// TIA Portal project "Sirius" (V17)

(* hardware
DEVICE "S7-1200 station_1"  S7-1200 Station
   slot 0: "Rack_0"  S7-1200 Rack  Rack  V1.0
   slot 1: "PLC_1"  CPU 1214C DC/DC/DC  6ES7 214-1AG40-0XB0  V4.5
   slot 2: "DI 16x24VDC/DQ 16xRelay_1"  SM 1223 DI16/DQ16 x relay  6ES7 223-1PL32-0XB0  V2.0
   slot 3: "DI 8/DQ 8x24VDC_1"  6ES7 223-1BH32-0XB0  V2.0
   slot 4: "AI 8x13BIT_1"  6ES7 231-4HF32-0XB0  V2.1
   slot 5: "AI 4x13BIT_1"  6ES7 231-4HD32-0XB0  V2.1
   slot 101: "CM 1241 (RS422/485)_1"  6ES7 241-1CH32-0XB0  V2.2
   slot 102: "CM 1241 (RS422/485)_2"  6ES7 241-1CH32-0XB0  V2.2
*)

// ===== PLC "PLC_1"  CPU 1214C DC/DC/DC =====

VAR_GLOBAL   // PLC tag table "Default tag table"
   "System_Byte" AT %MB1 : Byte;
   "FirstScan" AT %M1.0 : Bool;
   "DiagStatusUpdate" AT %M1.1 : Bool;
   "AlwaysTRUE" AT %M1.2 : Bool;
   "AlwaysFALSE" AT %M1.3 : Bool;
   "Clock_Byte" AT %MB0 : Byte;
   "Clock_10Hz" AT %M0.0 : Bool;
   "Clock_5Hz" AT %M0.1 : Bool;
   "Clock_2.5Hz" AT %M0.2 : Bool;
   "Clock_2Hz" AT %M0.3 : Bool;
   "Clock_1.25Hz" AT %M0.4 : Bool;
   "Clock_1Hz" AT %M0.5 : Bool;
   "Clock_0.625Hz" AT %M0.6 : Bool;
   "Clock_0.5Hz" AT %M0.7 : Bool;
END_VAR

VAR_GLOBAL   // PLC tag table "DI"
   "DIa1.0" AT %I0.0 : Bool;   // Наличие напряжения на основном вводе
   "DIa1.1" AT %I0.1 : Bool;   // Наличие напряжения на резервном вводе
   "DIa1.2" AT %I0.2 : Bool;   // Наличие питания 220В внешних потр.
   "DIa1.3" AT %I0.3 : Bool;   // Наличие пит. 220В собств. нужд; Питание 24В от АКБ
   "DIa1.4" AT %I0.4 : Bool;   // АКБ разряжена
   "DIa1.5" AT %I0.5 : Bool;   // Отключение звука
   "DIa1.6" AT %I0.6 : Bool;   // Стоп АН
   "DIa1.7" AT %I0.7 : Bool;   // Автоматическое управление
   "DIb1.0" AT %I1.0 : Bool;   // Ручное управление
   "DIb1.1" AT %I1.1 : Bool;   // Тест индикации
   "DIb1.2" AT %I1.2 : Bool;   // Затопление
   "DIb1.3" AT %I1.3 : Bool;   // Открытие двери
   "reserved_DIb1.4" AT %I1.4 : Bool;   // --------
   "reserved_DIb1.5" AT %I1.5 : Bool;   // --------
   "DIa2.0" AT %I8.0 : Bool;   // Авт. выкл. НБ № 1 включен
   "DIa2.1" AT %I8.1 : Bool;   // Контактор НБ № 1 вклюен
   "DIa2.2" AT %I8.2 : Bool;   // Авт. выкл. НБ № 2 включен
   "DIa2.3" AT %I8.3 : Bool;   // Контактор НБ № 2 включен
   "DIa2.4" AT %I8.4 : Bool;   // Авт. выкл. НБ № 3 включен
   "DIa2.5" AT %I8.5 : Bool;   // Контактор НБ № 3 включен
   "DIa2.6" AT %I8.6 : Bool;   // Авт. выкл. НБ № 4 включен
   "DIa2.7" AT %I8.7 : Bool;   // Контактор НБ № 4 включен
   "DIb2.0" AT %I9.0 : Bool;   // Авт. выкл. НБ № 5 включен
   "DIb2.1" AT %I9.1 : Bool;   // Контактор НБ № 5 включен
   "DIb2.2" AT %I9.2 : Bool;   // Авт. выкл. НП включен
   "DIb2.3" AT %I9.3 : Bool;   // Контактор НП включен
   "reserved_DIb2.4" AT %I9.4 : Bool;   // --------
   "reserved_DIb2.5" AT %I9.5 : Bool;   // --------
   "reserved_DIb2.6" AT %I9.6 : Bool;   // --------
   "reserved_DIb2.7" AT %I9.7 : Bool;   // --------
   "DIa3.0" AT %I12.0 : Bool;   // УУС.1: Проток
   "DIa3.1" AT %I12.1 : Bool;   // УУС.2: Проток
   "DIa3.2" AT %I12.2 : Bool;   // УУС.3: Проток
   "DIa3.3" AT %I12.3 : Bool;   // УУС.4: Проток
   "reserved_DIa3.4" AT %I12.4 : Bool;   // --------
   "reserved_DIa3.5" AT %I12.5 : Bool;   // --------
   "reserved_DIa3.6" AT %I12.6 : Bool;   // --------
   "reserved_DIa3.7" AT %I12.7 : Bool;   // --------
END_VAR

VAR_GLOBAL   // PLC tag table "DQ"
   "DQa1.0" AT %Q0.0 : Bool;   // Пожар
   "DQa1.1" AT %Q0.1 : Bool;   // Пуск насосного агрегата
   "DQa1.2" AT %Q0.2 : Bool;   // Отсутствие неисправности
   "DQa1.3" AT %Q0.3 : Bool;   // Автоматика отключена
   "DQa1.4" AT %Q0.4 : Bool;   // Дежурный режим
   "DQa1.5" AT %Q0.5 : Bool;   // Звуковой сигнал
   "DQa1.6" AT %Q0.6 : Bool;   // Система отключена
   "DQa1.7" AT %Q0.7 : Bool;   // Звук отключен
   "reserved_DQb1.0" AT %Q1.0 : Bool;   // -----
   "reserved_DQb1.1" AT %Q1.1 : Bool;   // -----
   "RQa2.0" AT %Q8.0 : Bool;   // Управление НБ № 1
   "RQa2.1" AT %Q8.1 : Bool;   // Управление НБ № 2
   "RQa2.2" AT %Q8.2 : Bool;   // Управление НБ № 3
   "RQa2.3" AT %Q8.3 : Bool;   // Управление НБ № 4
   "RQa2.4" AT %Q8.4 : Bool;   // Управление НБ № 5
   "RQa2.5" AT %Q8.5 : Bool;   // Управление НП
   "reserved_RQa2.6" AT %Q8.6 : Bool;   // -----
   "reserved_RQa2.7" AT %Q8.7 : Bool;   // -----
   "RQb2.0" AT %Q9.0 : Bool;   // Неисправность НБ № 1
   "RQb2.1" AT %Q9.1 : Bool;   // Неисправность НБ № 2
   "RQb2.2" AT %Q9.2 : Bool;   // Неисправность НБ № 3
   "RQb2.3" AT %Q9.3 : Bool;   // Неисправность НБ № 4
   "RQb2.4" AT %Q9.4 : Bool;   // Неисправность НБ № 5
   "RQb2.5" AT %Q9.5 : Bool;   // Неисправность НП
   "reserved_RQb2.6" AT %Q9.6 : Bool;   // -----
   "reserved_RQb2.7" AT %Q9.7 : Bool;   // -----
   "DQa3.0" AT %Q12.0 : Bool;   // УУС.1: Срабатывание
   "DQa3.1" AT %Q12.1 : Bool;   // УУС.1: Неисправность
   "DQa3.2" AT %Q12.2 : Bool;   // УУС.2: Срабатывание
   "DQa3.3" AT %Q12.3 : Bool;   // УУС.2: Неисправность
   "DQa3.4" AT %Q12.4 : Bool;   // УУС.3: Срабатывание
   "DQa3.5" AT %Q12.5 : Bool;   // УУС.3: Неисправность
   "DQa3.6" AT %Q12.6 : Bool;   // УУС.4: Срабатывание
   "DQa3.7" AT %Q12.7 : Bool;   // УУС.4: Неисправность
END_VAR

VAR_GLOBAL   // PLC tag table "AI"
   "AI4.0" AT %IW144 : Int;   // Датчик низкого давления PIS1.1
   "AI4.1" AT %IW146 : Int;   // Датчик низкого давления PIS1.2
   "AI4.2" AT %IW148 : Int;   // Датчик высокого давления PIS2.1
   "AI4.3" AT %IW150 : Int;   // Датчик высокого давления PIS2.2
   "AI4.4" AT %IW152 : Int;   // Датчик давления НБ №1
   "AI4.5" AT %IW154 : Int;   // Датчик давления НБ №2
   "AI4.6" AT %IW156 : Int;   // Датчик давления НБ №3
   "AI4.7" AT %IW158 : Int;   // Датчик давления НБ №4
   "AI5.0" AT %IW160 : Int;   // Датчик давления НБ №5
   "reserved_AI5.1" AT %IW162 : Int;   // ------
   "reserved_AI5.2" AT %IW164 : Int;   // ------
   "reserved_AI5.3" AT %IW166 : Int;   // ------
END_VAR

VAR_GLOBAL   // PLC tag table "MODBUS"
   "MB_MODE_auto" AT %M4002.1 : Bool;
   "MB_MODE_manual" AT %M4002.2 : Bool;
   "MB_MODE_blocked" AT %M4002.3 : Bool;
   "MB_MODE_standby" AT %M4002.4 : Bool;
   "MB_MODE_standby_pressure_high" AT %M4002.5 : Bool;
   "MB_BUTTON_Global_Stop" AT %M4002.6 : Bool;
   "MB_Global_Stop" AT %M4002.7 : Bool;
   "MB_BUTTON_Sound_Off" AT %M4003.0 : Bool;
   "MB_BUTTON_Led_Test" AT %M4003.1 : Bool;
   "MB_STATE_380_main" AT %M4003.2 : Bool;
   "MB_STATE_380_backup" AT %M4003.3 : Bool;
   "MB_STATE_220_inner" AT %M4003.4 : Bool;
   "MB_STATE_220_outer" AT %M4003.5 : Bool;
   "MB_STATE_door_opened" AT %M4003.6 : Bool;
   "MB_ERROR_underwater" AT %M4003.7 : Bool;
   "MB_ERROR_no_water" AT %M4004.0 : Bool;
   "MB_ERROR_no_water_fire" AT %M4004.1 : Bool;
   "MB_ERROR_inlet_pressure_low" AT %M4004.2 : Bool;
   "MB_ERROR_global" AT %M4004.3 : Bool;
   "MB_ERROR_Main_Ball_Valves" AT %M4004.4 : Bool;
   "MB_ERROR_BALL_VALVE_ANY" AT %M4004.5 : Bool;
   "MB_ERROR_any" AT %M4004.6 : Bool;
   "MB_SIGNAL_fire" AT %M4004.7 : Bool;
   "MB_SIGNAL_fire_by_pressure" AT %M4005.0 : Bool;
   "MB_ERROR_high_pressure_redundancy" AT %M4005.1 : Bool;
   "MB_ERROR_low_pressure_redundancy" AT %M4005.2 : Bool;
   "MB_SIGNAL_first_pump_has_started" AT %M4005.3 : Bool;
   "MB_Start_standby_pump" AT %M4005.4 : Bool;
   "MB_Secret_condition" AT %M4005.5 : Bool;
   "MB_ERROR_Battery_low" AT %M4005.6 : Bool;
   "MB_ERROR_connection_lost" AT %M4005.7 : Bool;
   "MB_ERROR_connection_lost_TOF" AT %M4006.0 : Bool;
   "MB_ERROR_connection_lost_TON" AT %M4006.1 : Bool;
   "MB_SENSOR_low_pressure_PIS1.1_error" AT %M4006.2 : Bool;
   "MB_SENSOR_low_pressure_PIS1.2_error" AT %M4006.3 : Bool;
   "MB_SENSOR_high_pressure_PIS2.1_error" AT %M4006.4 : Bool;
   "MB_SENSOR_high_pressure_PIS2.2_error" AT %M4006.5 : Bool;
   "MB_IN_valve_gate__ERROR_B1" AT %M4006.6 : Bool;
   "MB_IN_valve_gate__ERROR_B2" AT %M4006.7 : Bool;
   "MB_IN_valve_gate__ERROR_B3" AT %M4007.0 : Bool;
   "MB_IN_valve_gate__ERROR_B4" AT %M4007.1 : Bool;
   "MB_IN_valve_gate__ERROR_B5" AT %M4007.2 : Bool;
   "MB_IN_valve_gate__ERROR_B6" AT %M4007.3 : Bool;
   "MB_IN_valve_gate__ERROR_B7" AT %M4007.4 : Bool;
   "MB_IN_valve_gate__ERROR_B8" AT %M4007.5 : Bool;
   "MB_IN_valve_gate__ERROR_B9" AT %M4007.6 : Bool;
   "MB_ERROR_IN_VALVE_ANY" AT %M4007.7 : Bool;
   "MB_SENSOR_flow_UUS1" AT %M4008.0 : Bool;
   "MB_SENSOR_flow_UUS2" AT %M4008.1 : Bool;
   "MB_SENSOR_flow_UUS3" AT %M4008.2 : Bool;
   "MB_SENSOR_flow_UUS4" AT %M4008.3 : Bool;
   "MB_ERROR_UUS1" AT %M4008.4 : Bool;
   "MB_ERROR_UUS2" AT %M4008.5 : Bool;
   "MB_ERROR_UUS3" AT %M4008.6 : Bool;
   "MB_ERROR_UUS4" AT %M4008.7 : Bool;
   "MB_ERROR_UUS_ANY" AT %M4009.0 : Bool;
   "MB_ERROR_UUS_ALL" AT %M4009.1 : Bool;
   "MB_State_switch_pump1" AT %M4009.2 : Bool;
   "MB_State_switch_pump2" AT %M4009.3 : Bool;
   "MB_State_switch_pump3" AT %M4009.4 : Bool;
   "MB_State_switch_pump4" AT %M4009.5 : Bool;
   "MB_State_switch_pump5" AT %M4009.6 : Bool;
   "MB_Error_pump1" AT %M4009.7 : Bool;
   "MB_Error_pump2" AT %M4010.0 : Bool;
   "MB_Error_pump3" AT %M4010.1 : Bool;
   "MB_Error_pump4" AT %M4010.2 : Bool;
   "MB_Error_pump5" AT %M4010.3 : Bool;
   "MB_State_starter_pump1" AT %M4010.4 : Bool;
   "MB_State_starter_pump2" AT %M4010.5 : Bool;
   "MB_State_starter_pump3" AT %M4010.6 : Bool;
   "MB_State_starter_pump4" AT %M4010.7 : Bool;
   "MB_State_starter_pump5" AT %M4011.0 : Bool;
   "MB_State_work_pump1" AT %M4011.1 : Bool;
   "MB_State_work_pump2" AT %M4011.2 : Bool;
   "MB_State_work_pump3" AT %M4011.3 : Bool;
   "MB_State_work_pump4" AT %M4011.4 : Bool;
   "MB_State_work_pump5" AT %M4011.5 : Bool;
   "MB_Pump_pressure_sensor_error1" AT %M4011.6 : Bool;
   "MB_Pump_pressure_sensor_error2" AT %M4011.7 : Bool;
   "MB_Pump_pressure_sensor_error3" AT %M4012.0 : Bool;
   "MB_Pump_pressure_sensor_error4" AT %M4012.1 : Bool;
   "MB_Pump_pressure_sensor_error5" AT %M4012.2 : Bool;
   "MB_State_switch_standby_pump" AT %M4012.3 : Bool;
   "MB_Error_any_pump" AT %M4012.4 : Bool;
   "MB_Error_standby_pump" AT %M4012.5 : Bool;
   "MB_State_starter_standby_pump" AT %M4012.6 : Bool;
   "MB_State_work_standby_pump" AT %M4012.7 : Bool;
   "MB_State_work_any_pump" AT %M4013.0 : Bool;
   "MB_ERROR_PUMPS_ANY" AT %M4013.1 : Bool;
   "MB_ERROR_PUMPS_ALL" AT %M4013.2 : Bool;
   "MB_Low_pressure_valve_B1_open_OFF" AT %M4013.3 : Bool;
   "MB_Low_pressure_valve_B1_open_NO_signal" AT %M4013.4 : Bool;
   "MB_Low_pressure_valve_B1_open_short" AT %M4013.5 : Bool;
   "MB_Low_pressure_valve_B1_open_brake" AT %M4013.6 : Bool;
   "MB_Low_pressure_valve_B1_open_Signal" AT %M4013.7 : Bool;
   "MB_Low_pressure_valve_B1_close_OFF" AT %M4014.0 : Bool;
   "MB_Low_pressure_valve_B1_close_NO_signal" AT %M4014.1 : Bool;
   "MB_Low_pressure_valve_B1_close_short" AT %M4014.2 : Bool;
   "MB_Low_pressure_valve_B1_close_brake" AT %M4014.3 : Bool;
   "MB_Low_pressure_valve_B1_close_Signal" AT %M4014.4 : Bool;
   "MB_Low_pressure_valve_B2_open_OFF" AT %M4014.5 : Bool;
   "MB_Low_pressure_valve_B2_open_NO_signal" AT %M4014.6 : Bool;
   "MB_Low_pressure_valve_B2_open_short" AT %M4014.7 : Bool;
   "MB_Low_pressure_valve_B2_open_brake" AT %M4015.0 : Bool;
   "MB_Low_pressure_valve_B2_open_Signal" AT %M4015.1 : Bool;
   "MB_Low_pressure_valve_B2_close_OFF" AT %M4015.2 : Bool;
   "MB_Low_pressure_valve_B2_close_NO_signal" AT %M4015.3 : Bool;
   "MB_Low_pressure_valve_B2_close_short" AT %M4015.4 : Bool;
   "MB_Low_pressure_valve_B2_close_brake" AT %M4015.5 : Bool;
   "MB_Low_pressure_valve_B2_close_Signal" AT %M4015.6 : Bool;
   "MB_Low_pressure_valve_B3_open_OFF" AT %M4015.7 : Bool;
   "MB_Low_pressure_valve_B3_open_NO_signal" AT %M4016.0 : Bool;
   "MB_Low_pressure_valve_B3_open_short" AT %M4016.1 : Bool;
   "MB_Low_pressure_valve_B3_open_brake" AT %M4016.2 : Bool;
   "MB_Low_pressure_valve_B3_open_Signal" AT %M4016.3 : Bool;
   "MB_Low_pressure_valve_B3_close_OFF" AT %M4016.4 : Bool;
   "MB_Low_pressure_valve_B3_close_NO_signal" AT %M4016.5 : Bool;
   "MB_Low_pressure_valve_B3_close_short" AT %M4016.6 : Bool;
   "MB_Low_pressure_valve_B3_close_brake" AT %M4016.7 : Bool;
   "MB_Low_pressure_valve_B3_close_Signal" AT %M4017.0 : Bool;
   "MB_Low_pressure_valve_B4_open_OFF" AT %M4017.1 : Bool;
   "MB_Low_pressure_valve_B4_open_NO_signal" AT %M4017.2 : Bool;
   "MB_Low_pressure_valve_B4_open_short" AT %M4017.3 : Bool;
   "MB_Low_pressure_valve_B4_open_brake" AT %M4017.4 : Bool;
   "MB_Low_pressure_valve_B4_open_Signal" AT %M4017.5 : Bool;
   "MB_Low_pressure_valve_B4_close_OFF" AT %M4017.6 : Bool;
   "MB_Low_pressure_valve_B4_close_NO_signal" AT %M4017.7 : Bool;
   "MB_Low_pressure_valve_B4_close_short" AT %M4018.0 : Bool;
   "MB_Low_pressure_valve_B4_close_brake" AT %M4018.1 : Bool;
   "MB_Low_pressure_valve_B4_close_Signal" AT %M4018.2 : Bool;
   "MB_Low_pressure_valve_B5_open_OFF" AT %M4018.3 : Bool;
   "MB_Low_pressure_valve_B5_open_NO_signal" AT %M4018.4 : Bool;
   "MB_Low_pressure_valve_B5_open_short" AT %M4018.5 : Bool;
   "MB_Low_pressure_valve_B5_open_brake" AT %M4018.6 : Bool;
   "MB_Low_pressure_valve_B5_open_Signal" AT %M4018.7 : Bool;
   "MB_Low_pressure_valve_B5_close_OFF" AT %M4019.0 : Bool;
   "MB_Low_pressure_valve_B5_close_NO_signal" AT %M4019.1 : Bool;
   "MB_Low_pressure_valve_B5_close_short" AT %M4019.2 : Bool;
   "MB_Low_pressure_valve_B5_close_brake" AT %M4019.3 : Bool;
   "MB_Low_pressure_valve_B5_close_Signal" AT %M4019.4 : Bool;
   "MB_Low_pressure_valve_B6_open_OFF" AT %M4019.5 : Bool;
   "MB_Low_pressure_valve_B6_open_NO_signal" AT %M4019.6 : Bool;
   "MB_Low_pressure_valve_B6_open_short" AT %M4019.7 : Bool;
   "MB_Low_pressure_valve_B6_open_brake" AT %M4020.0 : Bool;
   "MB_Low_pressure_valve_B6_open_Signal" AT %M4020.1 : Bool;
   "MB_Low_pressure_valve_B6_close_OFF" AT %M4020.2 : Bool;
   "MB_Low_pressure_valve_B6_close_NO_signal" AT %M4020.3 : Bool;
   "MB_Low_pressure_valve_B6_close_short" AT %M4020.4 : Bool;
   "MB_Low_pressure_valve_B6_close_brake" AT %M4020.5 : Bool;
   "MB_Low_pressure_valve_B6_close_Signal" AT %M4020.6 : Bool;
   "MB_Low_pressure_valve_B7_open_OFF" AT %M4020.7 : Bool;
   "MB_Low_pressure_valve_B7_open_NO_signal" AT %M4021.0 : Bool;
   "MB_Low_pressure_valve_B7_open_short" AT %M4021.1 : Bool;
   "MB_Low_pressure_valve_B7_open_brake" AT %M4021.2 : Bool;
   "MB_Low_pressure_valve_B7_open_Signal" AT %M4021.3 : Bool;
   "MB_Low_pressure_valve_B7_close_OFF" AT %M4021.4 : Bool;
   "MB_Low_pressure_valve_B7_close_NO_signal" AT %M4021.5 : Bool;
   "MB_Low_pressure_valve_B7_close_short" AT %M4021.6 : Bool;
   "MB_Low_pressure_valve_B7_close_brake" AT %M4021.7 : Bool;
   "MB_Low_pressure_valve_B7_close_Signal" AT %M4022.0 : Bool;
   "MB_Low_pressure_valve_B8_open_OFF" AT %M4022.1 : Bool;
   "MB_Low_pressure_valve_B8_open_NO_signal" AT %M4022.2 : Bool;
   "MB_Low_pressure_valve_B8_open_short" AT %M4022.3 : Bool;
   "MB_Low_pressure_valve_B8_open_brake" AT %M4022.4 : Bool;
   "MB_Low_pressure_valve_B8_open_Signal" AT %M4022.5 : Bool;
   "MB_Low_pressure_valve_B8_close_OFF" AT %M4022.6 : Bool;
   "MB_Low_pressure_valve_B8_close_NO_signal" AT %M4022.7 : Bool;
   "MB_Low_pressure_valve_B8_close_short" AT %M4023.0 : Bool;
   "MB_Low_pressure_valve_B8_close_brake" AT %M4023.1 : Bool;
   "MB_Low_pressure_valve_B8_close_Signal" AT %M4023.2 : Bool;
   "MB_Low_pressure_valve_B9_open_OFF" AT %M4023.3 : Bool;
   "MB_Low_pressure_valve_B9_open_NO_signal" AT %M4023.4 : Bool;
   "MB_Low_pressure_valve_B9_open_short" AT %M4023.5 : Bool;
   "MB_Low_pressure_valve_B9_open_brake" AT %M4023.6 : Bool;
   "MB_Low_pressure_valve_B9_open_Signal" AT %M4023.7 : Bool;
   "MB_Low_pressure_valve_B9_close_OFF" AT %M4024.0 : Bool;
   "MB_Low_pressure_valve_B9_close_NO_signal" AT %M4024.1 : Bool;
   "MB_Low_pressure_valve_B9_close_short" AT %M4024.2 : Bool;
   "MB_Low_pressure_valve_B9_close_brake" AT %M4024.3 : Bool;
   "MB_Low_pressure_valve_B9_close_Signal" AT %M4024.4 : Bool;
   "MB_Ball_valve_K38.1_open_OFF" AT %M4024.5 : Bool;
   "MB_Ball_valve_K38.1_open_NO_signal" AT %M4024.6 : Bool;
   "MB_Ball_valve_K38.1_open_short" AT %M4024.7 : Bool;
   "MB_Ball_valve_K38.1_open_brake" AT %M4025.0 : Bool;
   "MB_Ball_valve_K38.1_open_Signal" AT %M4025.1 : Bool;
   "MB_Ball_valve_K38.2_open_OFF" AT %M4025.2 : Bool;
   "MB_Ball_valve_K38.2_open_NO_signal" AT %M4025.3 : Bool;
   "MB_Ball_valve_K38.2_open_short" AT %M4025.4 : Bool;
   "MB_Ball_valve_K38.2_open_brake" AT %M4025.5 : Bool;
   "MB_Ball_valve_K38.2_open_Signal" AT %M4025.6 : Bool;
   "MB_Ball_valve_K38.3_open_OFF" AT %M4025.7 : Bool;
   "MB_Ball_valve_K38.3_open_NO_signal" AT %M4026.0 : Bool;
   "MB_Ball_valve_K38.3_open_short" AT %M4026.1 : Bool;
   "MB_Ball_valve_K38.3_open_brake" AT %M4026.2 : Bool;
   "MB_Ball_valve_K38.3_open_Signal" AT %M4026.3 : Bool;
   "MB_Ball_valve_K38.4_open_OFF" AT %M4026.4 : Bool;
   "MB_Ball_valve_K38.4_open_NO_signal" AT %M4026.5 : Bool;
   "MB_Ball_valve_K38.4_open_short" AT %M4026.6 : Bool;
   "MB_Ball_valve_K38.4_open_brake" AT %M4026.7 : Bool;
   "MB_Ball_valve_K38.4_open_Signal" AT %M4027.0 : Bool;
   "MB_Ball_valve_K38.5_open_OFF" AT %M4027.1 : Bool;
   "MB_Ball_valve_K38.5_open_NO_signal" AT %M4027.2 : Bool;
   "MB_Ball_valve_K38.5_open_short" AT %M4027.3 : Bool;
   "MB_Ball_valve_K38.5_open_brake" AT %M4027.4 : Bool;
   "MB_Ball_valve_K38.5_open_Signal" AT %M4027.5 : Bool;
   "MB_UUS.1_open_OFF" AT %M4027.6 : Bool;
   "MB_UUS.1_open_NO_signal" AT %M4027.7 : Bool;
   "MB_UUS.1_open_short" AT %M4028.0 : Bool;
   "MB_UUS.1_open_brake" AT %M4028.1 : Bool;
   "MB_UUS.1_open_Signal" AT %M4028.2 : Bool;
   "MB_UUS.2_open_OFF" AT %M4028.3 : Bool;
   "MB_UUS.2_open_NO_signal" AT %M4028.4 : Bool;
   "MB_UUS.2_open_short" AT %M4028.5 : Bool;
   "MB_UUS.2_open_brake" AT %M4028.6 : Bool;
   "MB_UUS.2_open_Signal" AT %M4028.7 : Bool;
   "MB_UUS.3_open_OFF" AT %M4029.0 : Bool;
   "MB_UUS.3_open_NO_signal" AT %M4029.1 : Bool;
   "MB_UUS.3_open_short" AT %M4029.2 : Bool;
   "MB_UUS.3_open_brake" AT %M4029.3 : Bool;
   "MB_UUS.3_open_Signal" AT %M4029.4 : Bool;
   "MB_UUS.4_open_OFF" AT %M4029.5 : Bool;
   "MB_UUS.4_open_NO_signal" AT %M4029.6 : Bool;
   "MB_UUS.4_open_short" AT %M4029.7 : Bool;
   "MB_UUS.4_open_brake" AT %M4030.0 : Bool;
   "MB_UUS.4_open_Signal" AT %M4030.1 : Bool;
   "MB_SENSOR_low_pressure_PIS1.1" AT %MD4032 : Real;
   "MB_SENSOR_low_pressure_PIS1.2" AT %MD4036 : Real;
   "MB_SENSOR_high_pressure_PIS2.1" AT %MD4040 : Real;
   "MB_SENSOR_high_pressure_PIS2.2" AT %MD4044 : Real;
   "MB_INDICATION_high_pressure" AT %MD4048 : Real;
   "MB_INDICATION_low_pressure" AT %MD4052 : Real;
   "MB_Pump_pressure_sensor1" AT %MD4056 : Real;
   "MB_Pump_pressure_sensor2" AT %MD4060 : Real;
   "MB_Pump_pressure_sensor3" AT %MD4064 : Real;
   "MB_Pump_pressure_sensor4" AT %MD4068 : Real;
   "MB_Pump_pressure_sensor5" AT %MD4072 : Real;
   "MB_BUTTON_START_KPPU" AT %M4000.0 : Bool;
   "MB_BUTTON_STOP_KPPU" AT %M4000.1 : Bool;
   "MB_KPPU_connection_test" AT %M4000.2 : Bool;
   "MB_PPU_connection_test" AT %M4002.0 : Bool;
END_VAR

VAR_GLOBAL   // PLC tag table "HMI"
   "HMI_BUTTON_START_KPPU" AT %M600.0 : Bool;
   "HMI_BUTTON_STOP_KPPU" AT %M600.1 : Bool;
   "HMI_MODE_auto" AT %M600.2 : Bool;
   "HMI_MODE_manual" AT %M600.3 : Bool;
   "HMI_MODE_blocked" AT %M600.4 : Bool;
   "HMI_MODE_standby" AT %M600.5 : Bool;
   "HMI_MODE_standby_pressure_high" AT %M600.6 : Bool;
   "HMI_BUTTON_Global_Stop" AT %M600.7 : Bool;
   "HMI_Global_Stop" AT %M601.0 : Bool;
   "HMI_BUTTON_Sound_Off" AT %M601.1 : Bool;
   "HMI_BUTTON_Led_Test" AT %M601.2 : Bool;
   "HMI_STATE_380_main" AT %M601.3 : Bool;
   "HMI_STATE_380_backup" AT %M601.4 : Bool;
   "HMI_STATE_220_inner" AT %M601.5 : Bool;
   "HMI_STATE_220_outer" AT %M601.6 : Bool;
   "HMI_STATE_door_opened" AT %M601.7 : Bool;
   "HMI_ERROR_underwater" AT %M602.0 : Bool;
   "HMI_ERROR_no_water" AT %M602.1 : Bool;
   "HMI_ERROR_no_water_fire" AT %M602.2 : Bool;
   "HMI_ERROR_inlet_pressure_low" AT %M602.3 : Bool;
   "HMI_ERROR_global" AT %M602.4 : Bool;
   "HMI_ERROR_Main_Ball_Valves" AT %M602.5 : Bool;
   "HMI_ERROR_BALL_VALVE_ANY" AT %M602.6 : Bool;
   "HMI_ERROR_any" AT %M602.7 : Bool;
   "HMI_SIGNAL_fire" AT %M603.0 : Bool;
   "HMI_SIGNAL_fire_by_pressure" AT %M603.1 : Bool;
   "HMI_ERROR_high_pressure_redundancy" AT %M603.2 : Bool;
   "HMI_ERROR_low_pressure_redundancy" AT %M603.3 : Bool;
   "HMI_SIGNAL_first_pump_has_started" AT %M603.4 : Bool;
   "HMI_Start_standby_pump" AT %M603.5 : Bool;
   "HMI_Secret_condition" AT %M603.6 : Bool;
   "HMI_ERROR_Battery_low" AT %M603.7 : Bool;
   "HMI_ERROR_connection_lost" AT %M604.0 : Bool;
   "HMI_ERROR_connection_lost_TOF" AT %M604.1 : Bool;
   "HMI_ERROR_connection_lost_TON" AT %M604.2 : Bool;
   "HMI_SENSOR_low_pressure_PIS1.1_error" AT %M604.3 : Bool;
   "HMI_SENSOR_low_pressure_PIS1.2_error" AT %M604.4 : Bool;
   "HMI_SENSOR_high_pressure_PIS2.1_error" AT %M604.5 : Bool;
   "HMI_SENSOR_high_pressure_PIS2.2_error" AT %M604.6 : Bool;
   "HMI_IN_valve_gate__ERROR_B1" AT %M604.7 : Bool;
   "HMI_IN_valve_gate__ERROR_B2" AT %M605.0 : Bool;
   "HMI_IN_valve_gate__ERROR_B3" AT %M605.1 : Bool;
   "HMI_IN_valve_gate__ERROR_B4" AT %M605.2 : Bool;
   "HMI_IN_valve_gate__ERROR_B5" AT %M605.3 : Bool;
   "HMI_IN_valve_gate__ERROR_B6" AT %M605.4 : Bool;
   "HMI_IN_valve_gate__ERROR_B7" AT %M605.5 : Bool;
   "HMI_IN_valve_gate__ERROR_B8" AT %M605.6 : Bool;
   "HMI_IN_valve_gate__ERROR_B9" AT %M605.7 : Bool;
   "HMI_ERROR_IN_VALVE_ANY" AT %M606.0 : Bool;
   "HMI_SENSOR_flow_UUS1" AT %M606.1 : Bool;
   "HMI_SENSOR_flow_UUS2" AT %M606.2 : Bool;
   "HMI_SENSOR_flow_UUS3" AT %M606.3 : Bool;
   "HMI_SENSOR_flow_UUS4" AT %M606.4 : Bool;
   "HMI_ERROR_UUS1" AT %M606.5 : Bool;
   "HMI_ERROR_UUS2" AT %M606.6 : Bool;
   "HMI_ERROR_UUS3" AT %M606.7 : Bool;
   "HMI_ERROR_UUS4" AT %M607.0 : Bool;
   "HMI_ERROR_UUS_ANY" AT %M607.1 : Bool;
   "HMI_ERROR_UUS_ALL" AT %M607.2 : Bool;
   "HMI_State_switch_pump1" AT %M607.3 : Bool;
   "HMI_State_switch_pump2" AT %M607.4 : Bool;
   "HMI_State_switch_pump3" AT %M607.5 : Bool;
   "HMI_State_switch_pump4" AT %M607.6 : Bool;
   "HMI_State_switch_pump5" AT %M607.7 : Bool;
   "HMI_Error_pump1" AT %M608.0 : Bool;
   "HMI_Error_pump2" AT %M608.1 : Bool;
   "HMI_Error_pump3" AT %M608.2 : Bool;
   "HMI_Error_pump4" AT %M608.3 : Bool;
   "HMI_Error_pump5" AT %M608.4 : Bool;
   "HMI_State_starter_pump1" AT %M608.5 : Bool;
   "HMI_State_starter_pump2" AT %M608.6 : Bool;
   "HMI_State_starter_pump3" AT %M608.7 : Bool;
   "HMI_State_starter_pump4" AT %M609.0 : Bool;
   "HMI_State_starter_pump5" AT %M609.1 : Bool;
   "HMI_State_work_pump1" AT %M609.2 : Bool;
   "HMI_State_work_pump2" AT %M609.3 : Bool;
   "HMI_State_work_pump3" AT %M609.4 : Bool;
   "HMI_State_work_pump4" AT %M609.5 : Bool;
   "HMI_State_work_pump5" AT %M609.6 : Bool;
   "HMI_Pump_pressure_sensor_error1" AT %M609.7 : Bool;
   "HMI_Pump_pressure_sensor_error2" AT %M610.0 : Bool;
   "HMI_Pump_pressure_sensor_error3" AT %M610.1 : Bool;
   "HMI_Pump_pressure_sensor_error4" AT %M610.2 : Bool;
   "HMI_Pump_pressure_sensor_error5" AT %M610.3 : Bool;
   "HMI_State_switch_standby_pump" AT %M610.4 : Bool;
   "HMI_Error_any_pump" AT %M610.5 : Bool;
   "HMI_Error_standby_pump" AT %M610.6 : Bool;
   "HMI_State_starter_standby_pump" AT %M610.7 : Bool;
   "HMI_State_work_standby_pump" AT %M611.0 : Bool;
   "HMI_State_work_any_pump" AT %M611.1 : Bool;
   "HMI_ERROR_PUMPS_ANY" AT %M611.2 : Bool;
   "HMI_ERROR_PUMPS_ALL" AT %M611.3 : Bool;
   "HMI_Low_pressure_valve_B1_open_OFF" AT %M611.4 : Bool;
   "HMI_Low_pressure_valve_B1_open_NO_signal" AT %M611.5 : Bool;
   "HMI_Low_pressure_valve_B1_open_short" AT %M611.6 : Bool;
   "HMI_Low_pressure_valve_B1_open_brake" AT %M611.7 : Bool;
   "HMI_Low_pressure_valve_B1_open_Signal" AT %M612.0 : Bool;
   "HMI_Low_pressure_valve_B1_close_OFF" AT %M612.1 : Bool;
   "HMI_Low_pressure_valve_B1_close_NO_signal" AT %M612.2 : Bool;
   "HMI_Low_pressure_valve_B1_close_short" AT %M612.3 : Bool;
   "HMI_Low_pressure_valve_B1_close_brake" AT %M612.4 : Bool;
   "HMI_Low_pressure_valve_B1_close_Signal" AT %M612.5 : Bool;
   "HMI_Low_pressure_valve_B2_open_OFF" AT %M612.6 : Bool;
   "HMI_Low_pressure_valve_B2_open_NO_signal" AT %M612.7 : Bool;
   "HMI_Low_pressure_valve_B2_open_short" AT %M613.0 : Bool;
   "HMI_Low_pressure_valve_B2_open_brake" AT %M613.1 : Bool;
   "HMI_Low_pressure_valve_B2_open_Signal" AT %M613.2 : Bool;
   "HMI_Low_pressure_valve_B2_close_OFF" AT %M613.3 : Bool;
   "HMI_Low_pressure_valve_B2_close_NO_signal" AT %M613.4 : Bool;
   "HMI_Low_pressure_valve_B2_close_short" AT %M613.5 : Bool;
   "HMI_Low_pressure_valve_B2_close_brake" AT %M613.6 : Bool;
   "HMI_Low_pressure_valve_B2_close_Signal" AT %M613.7 : Bool;
   "HMI_Low_pressure_valve_B3_open_OFF" AT %M614.0 : Bool;
   "HMI_Low_pressure_valve_B3_open_NO_signal" AT %M614.1 : Bool;
   "HMI_Low_pressure_valve_B3_open_short" AT %M614.2 : Bool;
   "HMI_Low_pressure_valve_B3_open_brake" AT %M614.3 : Bool;
   "HMI_Low_pressure_valve_B3_open_Signal" AT %M614.4 : Bool;
   "HMI_Low_pressure_valve_B3_close_OFF" AT %M614.5 : Bool;
   "HMI_Low_pressure_valve_B3_close_NO_signal" AT %M614.6 : Bool;
   "HMI_Low_pressure_valve_B3_close_short" AT %M614.7 : Bool;
   "HMI_Low_pressure_valve_B3_close_brake" AT %M615.0 : Bool;
   "HMI_Low_pressure_valve_B3_close_Signal" AT %M615.1 : Bool;
   "HMI_Low_pressure_valve_B4_open_OFF" AT %M615.2 : Bool;
   "HMI_Low_pressure_valve_B4_open_NO_signal" AT %M615.3 : Bool;
   "HMI_Low_pressure_valve_B4_open_short" AT %M615.4 : Bool;
   "HMI_Low_pressure_valve_B4_open_brake" AT %M615.5 : Bool;
   "HMI_Low_pressure_valve_B4_open_Signal" AT %M615.6 : Bool;
   "HMI_Low_pressure_valve_B4_close_OFF" AT %M615.7 : Bool;
   "HMI_Low_pressure_valve_B4_close_NO_signal" AT %M616.0 : Bool;
   "HMI_Low_pressure_valve_B4_close_short" AT %M616.1 : Bool;
   "HMI_Low_pressure_valve_B4_close_brake" AT %M616.2 : Bool;
   "HMI_Low_pressure_valve_B4_close_Signal" AT %M616.3 : Bool;
   "HMI_Low_pressure_valve_B5_open_OFF" AT %M616.4 : Bool;
   "HMI_Low_pressure_valve_B5_open_NO_signal" AT %M616.5 : Bool;
   "HMI_Low_pressure_valve_B5_open_short" AT %M616.6 : Bool;
   "HMI_Low_pressure_valve_B5_open_brake" AT %M616.7 : Bool;
   "HMI_Low_pressure_valve_B5_open_Signal" AT %M617.0 : Bool;
   "HMI_Low_pressure_valve_B5_close_OFF" AT %M617.1 : Bool;
   "HMI_Low_pressure_valve_B5_close_NO_signal" AT %M617.2 : Bool;
   "HMI_Low_pressure_valve_B5_close_short" AT %M617.3 : Bool;
   "HMI_Low_pressure_valve_B5_close_brake" AT %M617.4 : Bool;
   "HMI_Low_pressure_valve_B5_close_Signal" AT %M617.5 : Bool;
   "HMI_Low_pressure_valve_B6_open_OFF" AT %M617.6 : Bool;
   "HMI_Low_pressure_valve_B6_open_NO_signal" AT %M617.7 : Bool;
   "HMI_Low_pressure_valve_B6_open_short" AT %M618.0 : Bool;
   "HMI_Low_pressure_valve_B6_open_brake" AT %M618.1 : Bool;
   "HMI_Low_pressure_valve_B6_open_Signal" AT %M618.2 : Bool;
   "HMI_Low_pressure_valve_B6_close_OFF" AT %M618.3 : Bool;
   "HMI_Low_pressure_valve_B6_close_NO_signal" AT %M618.4 : Bool;
   "HMI_Low_pressure_valve_B6_close_short" AT %M618.5 : Bool;
   "HMI_Low_pressure_valve_B6_close_brake" AT %M618.6 : Bool;
   "HMI_Low_pressure_valve_B6_close_Signal" AT %M618.7 : Bool;
   "HMI_Low_pressure_valve_B7_open_OFF" AT %M619.0 : Bool;
   "HMI_Low_pressure_valve_B7_open_NO_signal" AT %M619.1 : Bool;
   "HMI_Low_pressure_valve_B7_open_short" AT %M619.2 : Bool;
   "HMI_Low_pressure_valve_B7_open_brake" AT %M619.3 : Bool;
   "HMI_Low_pressure_valve_B7_open_Signal" AT %M619.4 : Bool;
   "HMI_Low_pressure_valve_B7_close_OFF" AT %M619.5 : Bool;
   "HMI_Low_pressure_valve_B7_close_NO_signal" AT %M619.6 : Bool;
   "HMI_Low_pressure_valve_B7_close_short" AT %M619.7 : Bool;
   "HMI_Low_pressure_valve_B7_close_brake" AT %M620.0 : Bool;
   "HMI_Low_pressure_valve_B7_close_Signal" AT %M620.1 : Bool;
   "HMI_Low_pressure_valve_B8_open_OFF" AT %M620.2 : Bool;
   "HMI_Low_pressure_valve_B8_open_NO_signal" AT %M620.3 : Bool;
   "HMI_Low_pressure_valve_B8_open_short" AT %M620.4 : Bool;
   "HMI_Low_pressure_valve_B8_open_brake" AT %M620.5 : Bool;
   "HMI_Low_pressure_valve_B8_open_Signal" AT %M620.6 : Bool;
   "HMI_Low_pressure_valve_B8_close_OFF" AT %M620.7 : Bool;
   "HMI_Low_pressure_valve_B8_close_NO_signal" AT %M621.0 : Bool;
   "HMI_Low_pressure_valve_B8_close_short" AT %M621.1 : Bool;
   "HMI_Low_pressure_valve_B8_close_brake" AT %M621.2 : Bool;
   "HMI_Low_pressure_valve_B8_close_Signal" AT %M621.3 : Bool;
   "HMI_Low_pressure_valve_B9_open_OFF" AT %M621.4 : Bool;
   "HMI_Low_pressure_valve_B9_open_NO_signal" AT %M621.5 : Bool;
   "HMI_Low_pressure_valve_B9_open_short" AT %M621.6 : Bool;
   "HMI_Low_pressure_valve_B9_open_brake" AT %M621.7 : Bool;
   "HMI_Low_pressure_valve_B9_open_Signal" AT %M622.0 : Bool;
   "HMI_Low_pressure_valve_B9_close_OFF" AT %M622.1 : Bool;
   "HMI_Low_pressure_valve_B9_close_NO_signal" AT %M622.2 : Bool;
   "HMI_Low_pressure_valve_B9_close_short" AT %M622.3 : Bool;
   "HMI_Low_pressure_valve_B9_close_brake" AT %M622.4 : Bool;
   "HMI_Low_pressure_valve_B9_close_Signal" AT %M622.5 : Bool;
   "HMI_Ball_valve_K38.1_open_OFF" AT %M622.6 : Bool;
   "HMI_Ball_valve_K38.1_open_NO_signal" AT %M622.7 : Bool;
   "HMI_Ball_valve_K38.1_open_short" AT %M623.0 : Bool;
   "HMI_Ball_valve_K38.1_open_brake" AT %M623.1 : Bool;
   "HMI_Ball_valve_K38.1_open_Signal" AT %M623.2 : Bool;
   "HMI_Ball_valve_K38.2_open_OFF" AT %M623.3 : Bool;
   "HMI_Ball_valve_K38.2_open_NO_signal" AT %M623.4 : Bool;
   "HMI_Ball_valve_K38.2_open_short" AT %M623.5 : Bool;
   "HMI_Ball_valve_K38.2_open_brake" AT %M623.6 : Bool;
   "HMI_Ball_valve_K38.2_open_Signal" AT %M623.7 : Bool;
   "HMI_Ball_valve_K38.3_open_OFF" AT %M624.0 : Bool;
   "HMI_Ball_valve_K38.3_open_NO_signal" AT %M624.1 : Bool;
   "HMI_Ball_valve_K38.3_open_short" AT %M624.2 : Bool;
   "HMI_Ball_valve_K38.3_open_brake" AT %M624.3 : Bool;
   "HMI_Ball_valve_K38.3_open_Signal" AT %M624.4 : Bool;
   "HMI_Ball_valve_K38.4_open_OFF" AT %M624.5 : Bool;
   "HMI_Ball_valve_K38.4_open_NO_signal" AT %M624.6 : Bool;
   "HMI_Ball_valve_K38.4_open_short" AT %M624.7 : Bool;
   "HMI_Ball_valve_K38.4_open_brake" AT %M625.0 : Bool;
   "HMI_Ball_valve_K38.4_open_Signal" AT %M625.1 : Bool;
   "HMI_Ball_valve_K38.5_open_OFF" AT %M625.2 : Bool;
   "HMI_Ball_valve_K38.5_open_NO_signal" AT %M625.3 : Bool;
   "HMI_Ball_valve_K38.5_open_short" AT %M625.4 : Bool;
   "HMI_Ball_valve_K38.5_open_brake" AT %M625.5 : Bool;
   "HMI_Ball_valve_K38.5_open_Signal" AT %M625.6 : Bool;
   "HMI_UUS.1_open_OFF" AT %M625.7 : Bool;
   "HMI_UUS.1_open_NO_signal" AT %M626.0 : Bool;
   "HMI_UUS.1_open_short" AT %M626.1 : Bool;
   "HMI_UUS.1_open_brake" AT %M626.2 : Bool;
   "HMI_UUS.1_open_Signal" AT %M626.3 : Bool;
   "HMI_UUS.2_open_OFF" AT %M626.4 : Bool;
   "HMI_UUS.2_open_NO_signal" AT %M626.5 : Bool;
   "HMI_UUS.2_open_short" AT %M626.6 : Bool;
   "HMI_UUS.2_open_brake" AT %M626.7 : Bool;
   "HMI_UUS.2_open_Signal" AT %M627.0 : Bool;
   "HMI_UUS.3_open_OFF" AT %M627.1 : Bool;
   "HMI_UUS.3_open_NO_signal" AT %M627.2 : Bool;
   "HMI_UUS.3_open_short" AT %M627.3 : Bool;
   "HMI_UUS.3_open_brake" AT %M627.4 : Bool;
   "HMI_UUS.3_open_Signal" AT %M627.5 : Bool;
   "HMI_UUS.4_open_OFF" AT %M627.6 : Bool;
   "HMI_UUS.4_open_NO_signal" AT %M627.7 : Bool;
   "HMI_UUS.4_open_short" AT %M628.0 : Bool;
   "HMI_UUS.4_open_brake" AT %M628.1 : Bool;
   "HMI_UUS.4_open_Signal" AT %M628.2 : Bool;
   "HMI_SENSOR_low_pressure_PIS1.1" AT %MD630 : Real;
   "HMI_SENSOR_low_pressure_PIS1.2" AT %MD634 : Real;
   "HMI_SENSOR_high_pressure_PIS2.1" AT %MD638 : Real;
   "HMI_SENSOR_high_pressure_PIS2.2" AT %MD642 : Real;
   "HMI_INDICATION_high_pressure" AT %MD646 : Real;
   "HMI_INDICATION_low_pressure" AT %MD650 : Real;
   "HMI_Pump_pressure_sensor1" AT %MD654 : Real;
   "HMI_Pump_pressure_sensor2" AT %MD658 : Real;
   "HMI_Pump_pressure_sensor3" AT %MD662 : Real;
   "HMI_Pump_pressure_sensor4" AT %MD666 : Real;
   "HMI_Pump_pressure_sensor5" AT %MD670 : Real;
END_VAR

VAR_GLOBAL   // PLC tag table "ModbusHoldingRegisters"
   "WriteHoldingRegister_00" AT %MW4002 : Word;
   "WriteHoldingRegister_01" AT %MW4004 : Word;
   "WriteHoldingRegister_02" AT %MW4006 : Word;
   "WriteHoldingRegister_03" AT %MW4008 : Word;
   "WriteHoldingRegister_04" AT %MW4010 : Word;
   "WriteHoldingRegister_05" AT %MW4012 : Word;
   "WriteHoldingRegister_06" AT %MW4014 : Word;
   "WriteHoldingRegister_07" AT %MW4016 : Word;
   "WriteHoldingRegister_08" AT %MW4018 : Word;
   "WriteHoldingRegister_09" AT %MW4020 : Word;
   "WriteHoldingRegister_10" AT %MW4022 : Word;
   "WriteHoldingRegister_11" AT %MW4024 : Word;
   "WriteHoldingRegister_12" AT %MW4026 : Word;
   "WriteHoldingRegister_13" AT %MW4028 : Word;
   "WriteHoldingRegister_14" AT %MW4030 : Word;
   "WriteHoldingRegister_15" AT %MW4032 : Word;
   "WriteHoldingRegister_16" AT %MW4034 : Word;
   "WriteHoldingRegister_18" AT %MW4038 : Word;
   "WriteHoldingRegister_19" AT %MW4040 : Word;
   "WriteHoldingRegister_20" AT %MW4042 : Word;
   "WriteHoldingRegister_22" AT %MW4046 : Word;
   "WriteHoldingRegister_23" AT %MW4048 : Word;
   "WriteHoldingRegister_24" AT %MW4050 : Word;
   "WriteHoldingRegister_25" AT %MW4052 : Word;
   "WriteHoldingRegister_26" AT %MW4054 : Word;
   "WriteHoldingRegister_27" AT %MW4056 : Word;
   "WriteHoldingRegister_28" AT %MW4058 : Word;
   "WriteHoldingRegister_29" AT %MW4060 : Word;
   "ReadHoldingRegister" AT %MW4000 : Word;
   "WriteHoldingRegister_17" AT %MW4036 : Word;
   "WriteHoldingRegister_21" AT %MW4044 : Word;
   "WriteHoldingRegister_30" AT %MW4062 : Word;
   "WriteHoldingRegister_31" AT %MW4064 : Word;
   "WriteHoldingRegister_32" AT %MW4066 : Word;
   "WriteHoldingRegister_33" AT %MW4068 : Word;
   "WriteHoldingRegister_34" AT %MW4070 : Word;
   "WriteHoldingRegister_35" AT %MW4072 : Word;
   "WriteHoldingRegister_36" AT %MW4074 : Word;
   "WriteHoldingRegister_37" AT %MW4076 : Word;
   "WriteHoldingRegister_38" AT %MW4078 : Word;
END_VAR

// folder: MAIN_DB

DATA_BLOCK "Section_valves_data"   // DB2
{ S7_Optimized_Access := 'TRUE' }
VERSION : 0.1
   VAR
      SENSOR_flow_UUS : Array[1..4] of Bool;
      ERROR_UUS : Array[1..4] of Bool;
      ERROR_UUS_ANY : Bool;
      ERROR_UUS_ALL : Bool;
   END_VAR
BEGIN
END_DATA_BLOCK

DATA_BLOCK "Preset_values"   // DB3
{ S7_Optimized_Access := 'TRUE' }
VERSION : 0.1
   VAR
      DI_timer_delay_time_superfast : Time := T#0.2s;
      DI_timer_delay_time_fast : Time := T#0.5s;
      DI_timer_delay_time_regular : Time := T#1s;
      DI_timer_delay_time_slow : Time := T#3s;
      DI_timer_delay_time_superslow : Time := T#5s;
      DI_timer_delay_time_gate_valve : Time := T#45s;
   END_VAR
BEGIN
END_DATA_BLOCK

DATA_BLOCK "Global"   // DB47
{ S7_Optimized_Access := 'TRUE' }
VERSION : 0.1
   VAR
      MODE_auto : Bool;
      MODE_manual : Bool;
      MODE_blocked : Bool;
      MODE_standby : Bool;
      MODE_standby_pressure_high : Bool;
      BUTTON_Global_Stop : Bool;
      Global_Stop : Bool;
      BUTTON_Sound_Off : Bool;
      BUTTON_Led_Test : Bool;
      STATE_380_main : Bool;
      STATE_380_backup : Bool;
      STATE_220_inner : Bool;
      STATE_220_outer : Bool;
      STATE_door_opened : Bool;
      ERROR_underwater : Bool;
      ERROR_no_water : Bool;
      ERROR_no_water_fire : Bool;
      ERROR_inlet_pressure_low : Bool;
      ERROR_global : Bool;
      ERROR_Main_Ball_Valves : Bool;
      ERROR_BALL_VALVE_ANY : Bool;
      ERROR_any : Bool;
      SIGNAL_fire : Bool;
      SIGNAL_fire_by_pressure : Bool;
      "SENSOR_low_pressure_PIS1.1" : Real;
      "SENSOR_low_pressure_PIS1.2" : Real;
      "SENSOR_high_pressure_PIS2.1" : Real := 0.0;
      "SENSOR_high_pressure_PIS2.2" : Real := 0.0;
      INDICATION_high_pressure : Real := 0.0;
      INDICATION_low_pressure : Real;
      ERROR_high_pressure_redundancy : Bool;
      ERROR_low_pressure_redundancy : Bool;
      SIGNAL_first_pump_has_started : Bool;
      Start_standby_pump : Bool;
      Secret_condition : Bool := false;
      ERROR_Battery_low : Bool;
      ERROR_connection_lost : Bool;
      ERROR_connection_lost_TOF : Bool;
      ERROR_connection_lost_TON : Bool;
      "SENSOR_low_pressure_PIS1.1_error" : Bool;
      "SENSOR_low_pressure_PIS1.2_error" : Bool;
      "SENSOR_high_pressure_PIS2.1_error" : Bool;
      "SENSOR_high_pressure_PIS2.2_error" : Bool;
   END_VAR
BEGIN
END_DATA_BLOCK

DATA_BLOCK "Low_pressure_valves"   // DB54
{ S7_Optimized_Access := 'TRUE' }
VERSION : 0.1
   VAR
      IN_valve_gate__ERROR_B : Array[1..9] of Bool;
      ERROR_IN_VALVE_ANY : Bool;
   END_VAR
BEGIN
END_DATA_BLOCK

DATA_BLOCK "Pumps_data"   // DB73
{ S7_Optimized_Access := 'TRUE' }
VERSION : 0.1
   VAR
      State_switch_pump : Array[1..10] of Bool;
      Error_pump : Array[1..10] of Bool;
      State_starter_pump : Array[1..10] of Bool;
      State_work_pump : Array[1..10] of Bool;
      Pump_run : Array[1..10] of Bool;
      Pump_pressure_sensor : Array[1..10] of Real;
      Pump_pressure_sensor_error : Array[1..10] of Bool;
      State_switch_standby_pump : Bool;
      Error_any_pump : Bool;
      Error_standby_pump : Bool;
      State_starter_standby_pump : Bool;
      State_work_standby_pump : Bool;
      State_work_any_pump : Bool;
      ERROR_PUMPS_ANY : Bool;
      ERROR_PUMPS_ALL : Bool;
      Pump_work_counter_arr : Array[1..10] of Int;
      pump_work_counter : Int;
   END_VAR
BEGIN
END_DATA_BLOCK

DATA_BLOCK "User_Defined"   // DB100
{ S7_Optimized_Access := 'TRUE' }
VERSION : 0.1
   VAR
      Pressure_stanby_pump_low : Real := 2.29;
      Pressure_stanby_pump_on : Real := 2.3;
      Pressure_stanby_pump_stop : Real := 2.5;
      Pressure_cascade_start : Real := 8.6;
      Pressure_cascade_stop : Real := 10.0;
      Pressure_pump_is_ok : Real := 0.3;
      Timer_cascade_start : Time := T#20s;
      Timer_standby_pump : Time := T#45s;
      Pump_error_time_by_pressure : Time := T#60s;
      Pressure_stanby_pump_error : Real := 3.5;
      "Yurich_blood-alcohol_ppm" : Real := 2.1;
   END_VAR
BEGIN
END_DATA_BLOCK

DATA_BLOCK "SOVA_Modbus_Input"   // DB136
{ S7_Optimized_Access := 'FALSE' }
VERSION : 0.1
   VAR
      SOVA : Array[1..3, 1..12] of Word;
      MB_Line : Array[1..3, 1..12, 0..7] of Bool;
   END_VAR
BEGIN
   // MB_Line[3,3,0] : Кран шаровой КР38.3 - канал отключен
   // MB_Line[3,3,1] : Кран шаровой КР38.3 - нет сигнала
   // MB_Line[3,3,2] : Кран шаровой КР38.3 - есть сигнал
   // MB_Line[3,3,3] : Кран шаровой КР38.3 - есть сигнал
   // MB_Line[3,3,4] : Кран шаровой КР38.3 - КЗ
   // MB_Line[3,3,5] : Кран шаровой КР38.3 - обрыв
   // MB_Line[3,3,6] : Кран шаровой КР38.3 - СИГНАЛ
   // MB_Line[3,3,7] : Кран шаровой КР38.3 - НЕИСПРАВНОСТЬ
   // MB_Line[3,4,0] : Кран шаровой КР38.4 - канал отключен
   // MB_Line[3,4,1] : Кран шаровой КР38.4 - нет сигнала
   // MB_Line[3,4,2] : Кран шаровой КР38.4 - есть сигнал
   // MB_Line[3,4,3] : Кран шаровой КР38.4 - есть сигнал
   // MB_Line[3,4,4] : Кран шаровой КР38.4 - КЗ
   // MB_Line[3,4,5] : Кран шаровой КР38.4 - обрыв
   // MB_Line[3,4,6] : Кран шаровой КР38.4 - СИГНАЛ
   // MB_Line[3,4,7] : Кран шаровой КР38.4 - НЕИСПРАВНОСТЬ
   // MB_Line[3,5,0] : Кран шаровой КР38.5 - канал отключен
   // MB_Line[3,5,1] : Кран шаровой КР38.5 - нет сигнала
   // MB_Line[3,5,2] : Кран шаровой КР38.5 - есть сигнал
   // MB_Line[3,5,3] : Кран шаровой КР38.5 - есть сигнал
   // MB_Line[3,5,4] : Кран шаровой КР38.5 - КЗ
   // MB_Line[3,5,5] : Кран шаровой КР38.5 - обрыв
   // MB_Line[3,5,6] : Кран шаровой КР38.5 - СИГНАЛ
   // MB_Line[3,5,7] : Кран шаровой КР38.5 - НЕИСПРАВНОСТЬ
   // MB_Line[3,6,0] : -------
   // MB_Line[3,6,1] : -------
   // MB_Line[3,6,2] : -------
   // MB_Line[3,6,3] : -------
   // MB_Line[3,6,4] : -------
   // MB_Line[3,6,5] : -------
   // MB_Line[3,6,6] : -------
   // MB_Line[3,6,7] : -------
   // MB_Line[3,7,0] : УУС.1 - канал отключен
   // MB_Line[3,7,1] : УУС.1 - нет сигнала
   // MB_Line[3,7,2] : УУС.1 - есть сигнал
   // MB_Line[3,7,3] : УУС.1 - есть сигнал
   // MB_Line[3,7,4] : УУС.1 - КЗ
   // MB_Line[3,7,5] : УУС.1 - обрыв
   // MB_Line[3,7,6] : УУС.1 - СИГНАЛ
   // MB_Line[3,7,7] : УУС.1 - НЕИСПРАВНОСТЬ
   // MB_Line[3,8,0] : УУС.2 - канал отключен
   // MB_Line[3,8,1] : УУС.2 - нет сигнала
   // MB_Line[3,8,2] : УУС.2 - есть сигнал
   // MB_Line[3,8,3] : УУС.2 - есть сигнал
   // MB_Line[3,8,4] : УУС.2 - КЗ
   // MB_Line[3,8,5] : УУС.2 - обрыв
   // MB_Line[3,8,6] : УУС.2 - СИГНАЛ
   // MB_Line[3,8,7] : УУС.2 - НЕИСПРАВНОСТЬ
   // MB_Line[3,9,0] : УУС.3 - канал отключен
   // MB_Line[3,9,1] : УУС.3 - нет сигнала
   // MB_Line[3,9,2] : УУС.3 - есть сигнал
   // MB_Line[3,9,3] : УУС.3 - есть сигнал
   // MB_Line[3,9,4] : УУС.3 - КЗ
   // MB_Line[3,9,5] : УУС.3 - обрыв
   // MB_Line[3,9,6] : УУС.3 - СИГНАЛ
   // MB_Line[3,9,7] : УУС.3 - НЕИСПРАВНОСТЬ
   // MB_Line[3,10,0] : УУС.4 - канал отключен
   // MB_Line[3,10,1] : УУС.4 - нет сигнала
   // MB_Line[3,10,2] : УУС.4 - есть сигнал
   // MB_Line[3,10,3] : УУС.4 - есть сигнал
   // MB_Line[3,10,4] : УУС.4 - КЗ
   // MB_Line[3,10,5] : УУС.4 - обрыв
   // MB_Line[3,10,6] : УУС.4 - СИГНАЛ
   // MB_Line[3,10,7] : УУС.4 - НЕИСПРАВНОСТЬ
   // MB_Line[3,11,0] : -------
   // MB_Line[3,11,1] : -------
   // MB_Line[3,11,2] : -------
   // MB_Line[3,11,3] : -------
   // MB_Line[3,11,4] : -------
   // MB_Line[3,11,5] : -------
   // MB_Line[3,11,6] : -------
   // MB_Line[3,11,7] : -------
   // MB_Line[3,12,0] : -------
   // MB_Line[3,12,1] : -------
   // MB_Line[3,12,2] : -------
   // MB_Line[3,12,3] : -------
   // MB_Line[3,12,4] : -------
   // MB_Line[3,12,5] : -------
   // MB_Line[3,12,6] : -------
   // MB_Line[3,12,7] : -------
   // MB_Line[1,5,0] : Диск. затвор В3 Открыт - канал отключен
   // MB_Line[1,5,1] : Диск. затвор В3 Открыт - нет сигнала
   // MB_Line[1,5,2] : Диск. затвор В3 Открыт - есть сигнал
   // MB_Line[1,5,3] : Диск. затвор В3 Открыт - есть сигнал
   // MB_Line[1,5,4] : Диск. затвор В3 Открыт - КЗ
   // MB_Line[1,5,5] : Диск. затвор В3 Открыт - обрыв
   // MB_Line[1,5,6] : Диск. затвор В3 Открыт - СИГНАЛ
   // MB_Line[1,5,7] : Диск. затвор В3 Открыт - НЕИСПРАВНОСТЬ
   // MB_Line[1,6,0] : Диск. затвор В3 Закрыт - канал отключен
   // MB_Line[1,6,1] : Диск. затвор В3 Закрыт - нет сигнала
   // MB_Line[1,6,2] : Диск. затвор В3 Закрыт - есть сигнал
   // MB_Line[1,6,3] : Диск. затвор В3 Закрыт - есть сигнал
   // MB_Line[1,6,4] : Диск. затвор В3 Закрыт - КЗ
   // MB_Line[1,6,5] : Диск. затвор В3 Закрыт - обрыв
   // MB_Line[1,6,6] : Диск. затвор В3 Закрыт - СИГНАЛ
   // MB_Line[1,6,7] : Диск. затвор В3 Закрыт - НЕИСПРАВНОСТЬ
   // MB_Line[1,7,0] : Диск. затвор В4 Открыт - канал отключен
   // MB_Line[1,7,1] : Диск. затвор В4 Открыт - нет сигнала
   // MB_Line[1,7,2] : Диск. затвор В4 Открыт - есть сигнал
   // MB_Line[1,7,3] : Диск. затвор В4 Открыт - есть сигнал
   // MB_Line[1,7,4] : Диск. затвор В4 Открыт - КЗ
   // MB_Line[1,7,5] : Диск. затвор В4 Открыт - обрыв
   // MB_Line[1,7,6] : Диск. затвор В4 Открыт - СИГНАЛ
   // MB_Line[1,7,7] : Диск. затвор В4 Открыт - НЕИСПРАВНОСТЬ
   // MB_Line[1,8,0] : Диск. затвор В4 Закрыт - канал отключен
   // MB_Line[1,8,1] : Диск. затвор В4 Закрыт - нет сигнала
   // MB_Line[1,8,2] : Диск. затвор В4 Закрыт - есть сигнал
   // MB_Line[1,8,3] : Диск. затвор В4 Закрыт - есть сигнал
   // MB_Line[1,8,4] : Диск. затвор В4 Закрыт - КЗ
   // MB_Line[1,8,5] : Диск. затвор В4 Закрыт - обрыв
   // MB_Line[1,8,6] : Диск. затвор В4 Закрыт - СИГНАЛ
   // MB_Line[1,8,7] : Диск. затвор В4 Закрыт - НЕИСПРАВНОСТЬ
   // MB_Line[1,9,0] : Диск. затвор В5 Открыт - канал отключен
   // MB_Line[1,9,1] : Диск. затвор В5 Открыт - нет сигнала
   // MB_Line[1,9,2] : Диск. затвор В5 Открыт - есть сигнал
   // MB_Line[1,9,3] : Диск. затвор В5 Открыт - есть сигнал
   // MB_Line[1,9,4] : Диск. затвор В5 Открыт - КЗ
   // MB_Line[1,9,5] : Диск. затвор В5 Открыт - обрыв
   // MB_Line[1,9,6] : Диск. затвор В5 Открыт - СИГНАЛ
   // MB_Line[1,9,7] : Диск. затвор В5 Открыт - НЕИСПРАВНОСТЬ
   // MB_Line[1,10,0] : Диск. затвор В5 Закрыт - канал отключен
   // MB_Line[1,10,1] : Диск. затвор В5 Закрыт - нет сигнала
   // MB_Line[1,10,2] : Диск. затвор В5 Закрыт - есть сигнал
   // MB_Line[1,10,3] : Диск. затвор В5 Закрыт - есть сигнал
   // MB_Line[1,10,4] : Диск. затвор В5 Закрыт - КЗ
   // MB_Line[1,10,5] : Диск. затвор В5 Закрыт - обрыв
   // MB_Line[1,10,6] : Диск. затвор В5 Закрыт - СИГНАЛ
   // MB_Line[1,10,7] : Диск. затвор В5 Закрыт - НЕИСПРАВНОСТЬ
   // MB_Line[1,11,1] : Диск. затвор В6 Открыт - нет сигнала
   // MB_Line[1,11,2] : Диск. затвор В6 Открыт - есть сигнал
   // MB_Line[1,11,0] : Диск. затвор В6 Открыт - канал отключен
   // MB_Line[1,11,3] : Диск. затвор В6 Открыт - есть сигнал
   // MB_Line[1,11,4] : Диск. затвор В6 Открыт - КЗ
   // MB_Line[1,11,5] : Диск. затвор В6 Открыт - обрыв
   // MB_Line[1,11,6] : Диск. затвор В6 Открыт - СИГНАЛ
   // MB_Line[1,11,7] : Диск. затвор В6 Открыт - НЕИСПРАВНОСТЬ
   // MB_Line[1,12,0] : Диск. затвор В6 Закрыт - канал отключен
   // MB_Line[1,12,1] : Диск. затвор В6 Закрыт - нет сигнала
   // MB_Line[1,12,2] : Диск. затвор В6 Закрыт - есть сигнал
   // MB_Line[1,12,3] : Диск. затвор В6 Закрыт - есть сигнал
   // MB_Line[1,12,4] : Диск. затвор В6 Закрыт - КЗ
   // MB_Line[1,12,5] : Диск. затвор В6 Закрыт - обрыв
   // MB_Line[1,12,6] : Диск. затвор В6 Закрыт - СИГНАЛ
   // MB_Line[1,12,7] : Диск. затвор В6 Закрыт - НЕИСПРАВНОСТЬ
   // MB_Line[2,1,0] : Диск. затвор В7 Открыт - канал отключен
   // MB_Line[2,1,1] : Диск. затвор В7 Открыт - нет сигнала
   // MB_Line[2,1,2] : Диск. затвор В7 Открыт - есть сигнал
   // MB_Line[2,1,3] : Диск. затвор В7 Открыт - есть сигнал
   // MB_Line[2,1,4] : Диск. затвор В7 Открыт - КЗ
   // MB_Line[2,1,5] : Диск. затвор В7 Открыт - обрыв
   // MB_Line[2,1,6] : Диск. затвор В7 Открыт - СИГНАЛ
   // MB_Line[2,1,7] : Диск. затвор В7 Открыт - НЕИСПРАВНОСТЬ
   // MB_Line[2,2,0] : Диск. затвор В7 Закрыт - канал отключен
   // MB_Line[2,2,1] : Диск. затвор В7 Закрыт - нет сигнала
   // MB_Line[2,2,2] : Диск. затвор В7 Закрыт - есть сигнал
   // MB_Line[2,2,3] : Диск. затвор В7 Закрыт - есть сигнал
   // MB_Line[2,2,4] : Диск. затвор В7 Закрыт - КЗ
   // MB_Line[2,2,5] : Диск. затвор В7 Закрыт - обрыв
   // MB_Line[2,2,6] : Диск. затвор В7 Закрыт - СИГНАЛ
   // MB_Line[2,2,7] : Диск. затвор В7 Закрыт - НЕИСПРАВНОСТЬ
   // MB_Line[2,3,0] : Диск. затвор В8 Открыт - канал отключен
   // MB_Line[2,3,1] : Диск. затвор В8 Открыт - нет сигнала
   // MB_Line[2,3,2] : Диск. затвор В8 Открыт - есть сигнал
   // MB_Line[2,3,3] : Диск. затвор В8 Открыт - есть сигнал
   // MB_Line[2,3,4] : Диск. затвор В8 Открыт - КЗ
   // MB_Line[2,3,5] : Диск. затвор В8 Открыт - обрыв
   // MB_Line[2,3,6] : Диск. затвор В8 Открыт - СИГНАЛ
   // MB_Line[2,3,7] : Диск. затвор В8 Открыт - НЕИСПРАВНОСТЬ
   // MB_Line[2,4,0] : Диск. затвор В8 Закрыт - канал отключен
   // MB_Line[2,4,1] : Диск. затвор В8 Закрыт - нет сигнала
   // MB_Line[2,4,2] : Диск. затвор В8 Закрыт - есть сигнал
   // MB_Line[2,4,3] : Диск. затвор В8 Закрыт - есть сигнал
   // MB_Line[2,4,4] : Диск. затвор В8 Закрыт - КЗ
   // MB_Line[2,4,5] : Диск. затвор В8 Закрыт - обрыв
   // MB_Line[2,4,6] : Диск. затвор В8 Закрыт - СИГНАЛ
   // MB_Line[2,4,7] : Диск. затвор В8 Закрыт - НЕИСПРАВНОСТЬ
   // MB_Line[2,5,0] : Диск. затвор В9 Открыт - канал отключен
   // MB_Line[2,5,1] : Диск. затвор В9 Открыт - нет сигнала
   // MB_Line[2,5,2] : Диск. затвор В9 Открыт - есть сигнал
   // MB_Line[2,5,3] : Диск. затвор В9 Открыт - есть сигнал
   // MB_Line[2,5,4] : Диск. затвор В9 Открыт - КЗ
   // MB_Line[2,5,5] : Диск. затвор В9 Открыт - обрыв
   // MB_Line[2,5,6] : Диск. затвор В9 Открыт - СИГНАЛ
   // MB_Line[2,5,7] : Диск. затвор В9 Открыт - НЕИСПРАВНОСТЬ
   // MB_Line[2,6,0] : Диск. затвор В9 Закрыт - канал отключен
   // MB_Line[2,6,1] : Диск. затвор В9 Закрыт - нет сигнала
   // MB_Line[2,6,2] : Диск. затвор В9 Закрыт - есть сигнал
   // MB_Line[2,6,3] : Диск. затвор В9 Закрыт - есть сигнал
   // MB_Line[2,6,4] : Диск. затвор В9 Закрыт - КЗ
   // MB_Line[2,6,5] : Диск. затвор В9 Закрыт - обрыв
   // MB_Line[2,6,6] : Диск. затвор В9 Закрыт - СИГНАЛ
   // MB_Line[2,6,7] : Диск. затвор В9 Закрыт - НЕИСПРАВНОСТЬ
   // MB_Line[2,11,0] : -------
   // MB_Line[2,11,1] : -------
   // MB_Line[2,11,2] : -------
   // MB_Line[2,11,3] : -------
   // MB_Line[2,11,4] : -------
   // MB_Line[2,11,5] : -------
   // MB_Line[2,11,6] : -------
   // MB_Line[2,11,7] : -------
   // MB_Line[2,12,0] : -------
   // MB_Line[2,12,1] : -------
   // MB_Line[2,12,2] : -------
   // MB_Line[2,12,3] : -------
   // MB_Line[2,12,4] : -------
   // MB_Line[2,12,5] : -------
   // MB_Line[2,12,6] : -------
   // MB_Line[2,12,7] : -------
   // MB_Line[3,1,0] : Кран шаровой КР38.1 - канал отключен
   // MB_Line[3,1,1] : Кран шаровой КР38.1 - нет сигнала
   // MB_Line[3,1,2] : Кран шаровой КР38.1 - есть сигнал
   // MB_Line[3,1,3] : Кран шаровой КР38.1 - есть сигнал
   // MB_Line[3,1,4] : Кран шаровой КР38.1 - КЗ
   // MB_Line[3,1,5] : Кран шаровой КР38.1 - обрыв
   // MB_Line[3,1,6] : Кран шаровой КР38.1 - СИГНАЛ
   // MB_Line[3,1,7] : Кран шаровой КР38.1 - НЕИСПРАВНОСТЬ
   // MB_Line[3,2,0] : Кран шаровой КР38.2 - канал отключен
   // MB_Line[3,2,1] : Кран шаровой КР38.2 - нет сигнала
   // MB_Line[3,2,2] : Кран шаровой КР38.2 - есть сигнал
   // MB_Line[3,2,3] : Кран шаровой КР38.2 - есть сигнал
   // MB_Line[3,2,4] : Кран шаровой КР38.2 - КЗ
   // MB_Line[3,2,5] : Кран шаровой КР38.2 - обрыв
   // MB_Line[3,2,6] : Кран шаровой КР38.2 - СИГНАЛ
   // MB_Line[3,2,7] : Кран шаровой КР38.2 - НЕИСПРАВНОСТЬ
   // MB_Line[1,1,0] : Диск. затвор В1 Открыта - канал отключен
   // MB_Line[1,1,1] : Диск. затвор В1 Открыта - нет сигнала
   // MB_Line[1,1,2] : Диск. затвор В1 Открыта - есть сигнал
   // MB_Line[1,1,3] : Диск. затвор В1 Открыта - есть сигнал
   // MB_Line[1,1,4] : Диск. затвор В1 Открыта - КЗ
   // MB_Line[1,1,5] : Диск. затвор В1 Открыта - обрыв
   // MB_Line[1,1,6] : Диск. затвор В1 Открыта - СИГНАЛ
   // MB_Line[1,1,7] : Диск. затвор В1 Открыта - НЕИСПРАВНОСТЬ
   // MB_Line[1,2,0] : Диск. затвор В1 Закрыта - канал отключен
   // MB_Line[1,2,1] : Диск. затвор В1 Закрыта - нет сигнала
   // MB_Line[1,2,2] : Диск. затвор В1 Закрыта - есть сигнал
   // MB_Line[1,2,3] : Диск. затвор В1 Закрыта - есть сигнал
   // MB_Line[1,2,4] : Диск. затвор В1 Закрыта - КЗ
   // MB_Line[1,2,5] : Диск. затвор В1 Закрыта - обрыв
   // MB_Line[1,2,6] : Диск. затвор В1 Закрыта - СИГНАЛ
   // MB_Line[1,2,7] : Диск. затвор В1 Закрыта - НЕИСПРАВНОСТЬ
   // MB_Line[1,3,0] : Диск. затвор В2 Открыта - канал отключен
   // MB_Line[1,3,1] : Диск. затвор В2 Открыта - нет сигнала
   // MB_Line[1,3,2] : Диск. затвор В2 Открыта - есть сигнал
   // MB_Line[1,3,3] : Диск. затвор В2 Открыта - есть сигнал
   // MB_Line[1,3,4] : Диск. затвор В2 Открыта - КЗ
   // MB_Line[1,3,5] : Диск. затвор В2 Открыта - обрыв
   // MB_Line[1,3,6] : Диск. затвор В2 Открыта - СИГНАЛ
   // MB_Line[1,3,7] : Диск. затвор В2 Открыта - НЕИСПРАВНОСТЬ
   // MB_Line[1,4,0] : Диск. затвор В2 Закрыта - канал отключен
   // MB_Line[1,4,1] : Диск. затвор В2 Закрыта - нет сигнала
   // MB_Line[1,4,2] : Диск. затвор В2 Закрыта - есть сигнал
   // MB_Line[1,4,3] : Диск. затвор В2 Закрыта - есть сигнал
   // MB_Line[1,4,4] : Диск. затвор В2 Закрыта - КЗ
   // MB_Line[1,4,5] : Диск. затвор В2 Закрыта - обрыв
   // MB_Line[1,4,6] : Диск. затвор В2 Закрыта - СИГНАЛ
   // MB_Line[1,4,7] : Диск. затвор В2 Закрыта - НЕИСПРАВНОСТЬ
   // MB_Line[2,7,0] : -------
   // MB_Line[2,7,1] : -------
   // MB_Line[2,7,2] : -------
   // MB_Line[2,7,3] : -------
   // MB_Line[2,7,4] : -------
   // MB_Line[2,7,5] : -------
   // MB_Line[2,7,6] : -------
   // MB_Line[2,7,7] : -------
   // MB_Line[2,8,0] : -------
   // MB_Line[2,8,1] : -------
   // MB_Line[2,8,2] : -------
   // MB_Line[2,8,3] : -------
   // MB_Line[2,8,4] : -------
   // MB_Line[2,8,5] : -------
   // MB_Line[2,8,6] : -------
   // MB_Line[2,8,7] : -------
   // MB_Line[2,9,0] : -------
   // MB_Line[2,9,1] : -------
   // MB_Line[2,9,2] : -------
   // MB_Line[2,9,3] : -------
   // MB_Line[2,9,4] : -------
   // MB_Line[2,9,5] : -------
   // MB_Line[2,9,6] : -------
   // MB_Line[2,9,7] : -------
   // MB_Line[2,10,0] : -------
   // MB_Line[2,10,1] : -------
   // MB_Line[2,10,2] : -------
   // MB_Line[2,10,4] : -------
   // MB_Line[2,10,3] : -------
   // MB_Line[2,10,5] : -------
   // MB_Line[2,10,6] : -------
   // MB_Line[2,10,7] : -------
END_DATA_BLOCK

// folder: Support_DB

DATA_BLOCK "State_380_main"   // DB1
{ S7_Optimized_Access := 'TRUE' }
VERSION : 0.1
// stored: InstanceOfName DI_Single
"DI_Single"
BEGIN
END_DATA_BLOCK

DATA_BLOCK "State_380_backup"   // DB4
{ S7_Optimized_Access := 'TRUE' }
VERSION : 0.1
// stored: InstanceOfName DI_Single
"DI_Single"
BEGIN
END_DATA_BLOCK

DATA_BLOCK "State_220_outer"   // DB5
{ S7_Optimized_Access := 'TRUE' }
VERSION : 0.1
// stored: InstanceOfName DI_Single
"DI_Single"
BEGIN
END_DATA_BLOCK

DATA_BLOCK "State_220_inner"   // DB6
{ S7_Optimized_Access := 'TRUE' }
VERSION : 0.1
// stored: InstanceOfName DI_Single
"DI_Single"
BEGIN
END_DATA_BLOCK

DATA_BLOCK "State_battery_low"   // DB7
{ S7_Optimized_Access := 'TRUE' }
VERSION : 0.1
// stored: InstanceOfName DI_Single
"DI_Single"
BEGIN
END_DATA_BLOCK

DATA_BLOCK "State_mode_auto"   // DB8
{ S7_Optimized_Access := 'TRUE' }
VERSION : 0.1
// stored: InstanceOfName DI_Single
"DI_Single"
BEGIN
END_DATA_BLOCK

DATA_BLOCK "State_mode_manual"   // DB9
{ S7_Optimized_Access := 'TRUE' }
VERSION : 0.1
// stored: InstanceOfName DI_Single
"DI_Single"
BEGIN
END_DATA_BLOCK

DATA_BLOCK "State_underwater"   // DB10
{ S7_Optimized_Access := 'TRUE' }
VERSION : 0.1
// stored: InstanceOfName DI_Single
"DI_Single"
BEGIN
END_DATA_BLOCK

DATA_BLOCK "State_door_opened"   // DB11
{ S7_Optimized_Access := 'TRUE' }
VERSION : 0.1
// stored: InstanceOfName DI_Single
"DI_Single"
BEGIN
END_DATA_BLOCK

DATA_BLOCK "Button_sound_off"   // DB12
{ S7_Optimized_Access := 'TRUE' }
VERSION : 0.1
// stored: InstanceOfName DI_Single
"DI_Single"
BEGIN
END_DATA_BLOCK

DATA_BLOCK "Button_global_stop"   // DB13
{ S7_Optimized_Access := 'TRUE' }
VERSION : 0.1
// stored: InstanceOfName DI_Single
"DI_Single"
BEGIN
END_DATA_BLOCK

DATA_BLOCK "Button_led_test"   // DB14
{ S7_Optimized_Access := 'TRUE' }
VERSION : 0.1
// stored: InstanceOfName DI_Single
"DI_Single"
BEGIN
END_DATA_BLOCK

DATA_BLOCK "State_switch_pump_1"   // DB15
{ S7_Optimized_Access := 'TRUE' }
VERSION : 0.1
// stored: InstanceOfName DI_Single
"DI_Single"
BEGIN
END_DATA_BLOCK

DATA_BLOCK "State_switch_pump_2"   // DB16
{ S7_Optimized_Access := 'TRUE' }
VERSION : 0.1
// stored: InstanceOfName DI_Single
"DI_Single"
BEGIN
END_DATA_BLOCK

DATA_BLOCK "State_switch_pump_3"   // DB17
{ S7_Optimized_Access := 'TRUE' }
VERSION : 0.1
// stored: InstanceOfName DI_Single
"DI_Single"
BEGIN
END_DATA_BLOCK

DATA_BLOCK "State_switch_pump_4"   // DB18
{ S7_Optimized_Access := 'TRUE' }
VERSION : 0.1
// stored: InstanceOfName DI_Single
"DI_Single"
BEGIN
END_DATA_BLOCK

DATA_BLOCK "State_switch_pump_5"   // DB19
{ S7_Optimized_Access := 'TRUE' }
VERSION : 0.1
// stored: InstanceOfName DI_Single
"DI_Single"
BEGIN
END_DATA_BLOCK

DATA_BLOCK "State_starter_pump_1"   // DB20
{ S7_Optimized_Access := 'TRUE' }
VERSION : 0.1
// stored: InstanceOfName DI_Single
"DI_Single"
BEGIN
END_DATA_BLOCK

DATA_BLOCK "State_starter_pump_2"   // DB21
{ S7_Optimized_Access := 'TRUE' }
VERSION : 0.1
// stored: InstanceOfName DI_Single
"DI_Single"
BEGIN
END_DATA_BLOCK

DATA_BLOCK "State_starter_pump_3"   // DB22
{ S7_Optimized_Access := 'TRUE' }
VERSION : 0.1
// stored: InstanceOfName DI_Single
"DI_Single"
BEGIN
END_DATA_BLOCK

DATA_BLOCK "State_starter_pump_4"   // DB23
{ S7_Optimized_Access := 'TRUE' }
VERSION : 0.1
// stored: InstanceOfName DI_Single
"DI_Single"
BEGIN
END_DATA_BLOCK

DATA_BLOCK "State_starter_pump_5"   // DB24
{ S7_Optimized_Access := 'TRUE' }
VERSION : 0.1
// stored: InstanceOfName DI_Single
"DI_Single"
BEGIN
END_DATA_BLOCK

DATA_BLOCK "State_switch_standby_pump"   // DB25
{ S7_Optimized_Access := 'TRUE' }
VERSION : 0.1
// stored: InstanceOfName DI_Single
"DI_Single"
BEGIN
END_DATA_BLOCK

DATA_BLOCK "State_starter_standby_pump"   // DB26
{ S7_Optimized_Access := 'TRUE' }
VERSION : 0.1
// stored: InstanceOfName DI_Single
"DI_Single"
BEGIN
END_DATA_BLOCK

DATA_BLOCK "State_UUS1_flow"   // DB27
{ S7_Optimized_Access := 'TRUE' }
VERSION : 0.1
// stored: InstanceOfName DI_Single
"DI_Single"
BEGIN
END_DATA_BLOCK

DATA_BLOCK "State_UUS2_flow"   // DB28
{ S7_Optimized_Access := 'TRUE' }
VERSION : 0.1
// stored: InstanceOfName DI_Single
"DI_Single"
BEGIN
END_DATA_BLOCK

DATA_BLOCK "State_UUS3_flow"   // DB29
{ S7_Optimized_Access := 'TRUE' }
VERSION : 0.1
// stored: InstanceOfName DI_Single
"DI_Single"
BEGIN
END_DATA_BLOCK

DATA_BLOCK "State_UUS4_flow"   // DB30
{ S7_Optimized_Access := 'TRUE' }
VERSION : 0.1
// stored: InstanceOfName DI_Single
"DI_Single"
BEGIN
END_DATA_BLOCK

DATA_BLOCK "Sound_1_DB"   // DB31
{ S7_Optimized_Access := 'TRUE' }
VERSION : 0.1
// stored: InstanceOfName Sound_PTO
"Sound_PTO"
BEGIN
END_DATA_BLOCK

DATA_BLOCK "ModbusMasterConnector_DB"   // DB33
{ S7_Optimized_Access := 'FALSE' }
VERSION : 0.1
// stored: InstanceOfName ModbusMasterConnector
"ModbusMasterConnector"
BEGIN
END_DATA_BLOCK

DATA_BLOCK "SOVA_Modbus_Input_Reading_DB"   // DB34
{ S7_Optimized_Access := 'TRUE' }
VERSION : 0.1
// stored: InstanceOfName SOVA_Modbus_Input_Reading
"SOVA_Modbus_Input_Reading"
BEGIN
END_DATA_BLOCK

DATA_BLOCK "State_work_pump_DB"   // DB38
{ S7_Optimized_Access := 'TRUE' }
VERSION : 0.1
// stored: InstanceOfName State_work_pump
"State_work_pump"
BEGIN
END_DATA_BLOCK

DATA_BLOCK "First_pump_start_DB"   // DB40
{ S7_Optimized_Access := 'TRUE' }
VERSION : 0.1
// stored: InstanceOfName First_pump_start
"First_pump_start"
BEGIN
END_DATA_BLOCK

DATA_BLOCK "Cascade_DB"   // DB43
{ S7_Optimized_Access := 'TRUE' }
VERSION : 0.1
// stored: InstanceOfName Cascade
"Cascade"
BEGIN
END_DATA_BLOCK

DATA_BLOCK "PumpRun_1"   // DB44
{ S7_Optimized_Access := 'TRUE' }
VERSION : 0.1
// stored: InstanceOfName PumpRun
"PumpRun"
BEGIN
END_DATA_BLOCK

DATA_BLOCK "PumpRun_2"   // DB45
{ S7_Optimized_Access := 'TRUE' }
VERSION : 0.1
// stored: InstanceOfName PumpRun
"PumpRun"
BEGIN
END_DATA_BLOCK

DATA_BLOCK "PumpRun_3"   // DB46
{ S7_Optimized_Access := 'TRUE' }
VERSION : 0.1
// stored: InstanceOfName PumpRun
"PumpRun"
BEGIN
END_DATA_BLOCK

DATA_BLOCK "PumpRun_4"   // DB48
{ S7_Optimized_Access := 'TRUE' }
VERSION : 0.1
// stored: InstanceOfName PumpRun
"PumpRun"
BEGIN
END_DATA_BLOCK

DATA_BLOCK "PumpRun_5"   // DB49
{ S7_Optimized_Access := 'TRUE' }
VERSION : 0.1
// stored: InstanceOfName PumpRun
"PumpRun"
BEGIN
END_DATA_BLOCK

DATA_BLOCK "Gate_Valve_Error_DB_B1"   // DB51
{ S7_Optimized_Access := 'TRUE' }
VERSION : 0.1
// stored: InstanceOfName Gate_Valve_Error
"Gate_Valve_Error"
BEGIN
END_DATA_BLOCK

DATA_BLOCK "Gate_Valve_Error_DB_B2"   // DB52
{ S7_Optimized_Access := 'TRUE' }
VERSION : 0.1
// stored: InstanceOfName Gate_Valve_Error
"Gate_Valve_Error"
BEGIN
END_DATA_BLOCK

DATA_BLOCK "Gate_Valve_Error_DB_B3"   // DB53
{ S7_Optimized_Access := 'TRUE' }
VERSION : 0.1
// stored: InstanceOfName Gate_Valve_Error
"Gate_Valve_Error"
BEGIN
END_DATA_BLOCK

DATA_BLOCK "Gate_Valve_Error_DB_B4"   // DB55
{ S7_Optimized_Access := 'TRUE' }
VERSION : 0.1
// stored: InstanceOfName Gate_Valve_Error
"Gate_Valve_Error"
BEGIN
END_DATA_BLOCK

DATA_BLOCK "Gate_Valve_Error_DB_B5"   // DB56
{ S7_Optimized_Access := 'TRUE' }
VERSION : 0.1
// stored: InstanceOfName Gate_Valve_Error
"Gate_Valve_Error"
BEGIN
END_DATA_BLOCK

DATA_BLOCK "Gate_Valve_Error_DB_B6"   // DB57
{ S7_Optimized_Access := 'TRUE' }
VERSION : 0.1
// stored: InstanceOfName Gate_Valve_Error
"Gate_Valve_Error"
BEGIN
END_DATA_BLOCK

DATA_BLOCK "Gate_Valve_Error_DB_B7"   // DB58
{ S7_Optimized_Access := 'TRUE' }
VERSION : 0.1
// stored: InstanceOfName Gate_Valve_Error
"Gate_Valve_Error"
BEGIN
END_DATA_BLOCK

DATA_BLOCK "Gate_Valve_Error_DB_B8"   // DB59
{ S7_Optimized_Access := 'TRUE' }
VERSION : 0.1
// stored: InstanceOfName Gate_Valve_Error
"Gate_Valve_Error"
BEGIN
END_DATA_BLOCK

DATA_BLOCK "Gate_Valve_Error_DB_B9"   // DB60
{ S7_Optimized_Access := 'TRUE' }
VERSION : 0.1
// stored: InstanceOfName Gate_Valve_Error
"Gate_Valve_Error"
BEGIN
END_DATA_BLOCK

DATA_BLOCK "Standby_Pump_Error_DB"   // DB61
{ S7_Optimized_Access := 'TRUE' }
VERSION : 0.1
// stored: InstanceOfName Standby_Pump/Compressor_Error
"Standby_Pump/Compressor_Error"
BEGIN
END_DATA_BLOCK

DATA_BLOCK "Pump_Error_1"   // DB62
{ S7_Optimized_Access := 'TRUE' }
VERSION : 0.1
// stored: InstanceOfName Pump_Error
"Pump_Error"
BEGIN
END_DATA_BLOCK

DATA_BLOCK "Pump_Error_2"   // DB63
{ S7_Optimized_Access := 'TRUE' }
VERSION : 0.1
// stored: InstanceOfName Pump_Error
"Pump_Error"
BEGIN
END_DATA_BLOCK

DATA_BLOCK "Pump_Error_3"   // DB64
{ S7_Optimized_Access := 'TRUE' }
VERSION : 0.1
// stored: InstanceOfName Pump_Error
"Pump_Error"
BEGIN
END_DATA_BLOCK

DATA_BLOCK "Pump_Error_4"   // DB65
{ S7_Optimized_Access := 'TRUE' }
VERSION : 0.1
// stored: InstanceOfName Pump_Error
"Pump_Error"
BEGIN
END_DATA_BLOCK

DATA_BLOCK "Pump_Error_5"   // DB66
{ S7_Optimized_Access := 'TRUE' }
VERSION : 0.1
// stored: InstanceOfName Pump_Error
"Pump_Error"
BEGIN
END_DATA_BLOCK

DATA_BLOCK "AI_Sensor_PIS1.1"   // DB67
{ S7_Optimized_Access := 'TRUE' }
VERSION : 0.1
// stored: InstanceOfName AI_Sensor
"AI_Sensor"
BEGIN
END_DATA_BLOCK

DATA_BLOCK "AI_Sensor_PIS1.2"   // DB68
{ S7_Optimized_Access := 'TRUE' }
VERSION : 0.1
// stored: InstanceOfName AI_Sensor
"AI_Sensor"
BEGIN
END_DATA_BLOCK

DATA_BLOCK "AI_Redundancy_low_pressure"   // DB69
{ S7_Optimized_Access := 'TRUE' }
VERSION : 0.1
// stored: InstanceOfName AI_Redundancy
"AI_Redundancy"
BEGIN
END_DATA_BLOCK

DATA_BLOCK "AI_Sensor_PIS2.1"   // DB70
{ S7_Optimized_Access := 'TRUE' }
VERSION : 0.1
// stored: InstanceOfName AI_Sensor
"AI_Sensor"
BEGIN
END_DATA_BLOCK

DATA_BLOCK "AI_Sensor_PIS2.2"   // DB71
{ S7_Optimized_Access := 'TRUE' }
VERSION : 0.1
// stored: InstanceOfName AI_Sensor
"AI_Sensor"
BEGIN
END_DATA_BLOCK

DATA_BLOCK "AI_Redundancy_high_pressure"   // DB72
{ S7_Optimized_Access := 'TRUE' }
VERSION : 0.1
// stored: InstanceOfName AI_Redundancy
"AI_Redundancy"
BEGIN
END_DATA_BLOCK

DATA_BLOCK "AI_Sensor_pump_1"   // DB74
{ S7_Optimized_Access := 'TRUE' }
VERSION : 0.1
// stored: InstanceOfName AI_Sensor
"AI_Sensor"
BEGIN
END_DATA_BLOCK

DATA_BLOCK "AI_Sensor_pump_2"   // DB75
{ S7_Optimized_Access := 'TRUE' }
VERSION : 0.1
// stored: InstanceOfName AI_Sensor
"AI_Sensor"
BEGIN
END_DATA_BLOCK

DATA_BLOCK "AI_Sensor_pump_3"   // DB76
{ S7_Optimized_Access := 'TRUE' }
VERSION : 0.1
// stored: InstanceOfName AI_Sensor
"AI_Sensor"
BEGIN
END_DATA_BLOCK

DATA_BLOCK "AI_Sensor_pump_4"   // DB77
{ S7_Optimized_Access := 'TRUE' }
VERSION : 0.1
// stored: InstanceOfName AI_Sensor
"AI_Sensor"
BEGIN
END_DATA_BLOCK

DATA_BLOCK "AI_Sensor_pump_5"   // DB78
{ S7_Optimized_Access := 'TRUE' }
VERSION : 0.1
// stored: InstanceOfName AI_Sensor
"AI_Sensor"
BEGIN
END_DATA_BLOCK

// folder: System blocks/Program resources

DATA_BLOCK "Timer_connection_test_1"   // DB35
{ S7_Optimized_Access := 'TRUE' }
AUTHOR : Simatic
FAMILY : IEC
NAME : IEC_TMR
VERSION : 1.0
// stored: InstanceOfName IEC_TIMER
"IEC_TIMER"
BEGIN
END_DATA_BLOCK

DATA_BLOCK "TImer_connection_test_2"   // DB36
{ S7_Optimized_Access := 'TRUE' }
AUTHOR : Simatic
FAMILY : IEC
NAME : IEC_TMR
VERSION : 1.0
// stored: InstanceOfName IEC_TIMER
"IEC_TIMER"
BEGIN
END_DATA_BLOCK

DATA_BLOCK "Timer_standby_pump"   // DB37
{ S7_Optimized_Access := 'TRUE' }
AUTHOR : Simatic
FAMILY : IEC
NAME : IEC_TMR
VERSION : 1.0
// stored: InstanceOfName IEC_TIMER
"IEC_TIMER"
BEGIN
END_DATA_BLOCK

DATA_BLOCK "IEC_Timer_0_DB_0"   // DB39
{ S7_Optimized_Access := 'TRUE' }
AUTHOR : Simatic
FAMILY : IEC
NAME : IEC_TMR
VERSION : 1.0
// stored: InstanceOfName IEC_TIMER
"IEC_TIMER"
BEGIN
END_DATA_BLOCK

DATA_BLOCK "IEC_Timer_0_DB_1"   // DB41
{ S7_Optimized_Access := 'TRUE' }
AUTHOR : Simatic
FAMILY : IEC
NAME : IEC_TMR
VERSION : 1.0
// stored: InstanceOfName IEC_TIMER
"IEC_TIMER"
BEGIN
END_DATA_BLOCK

DATA_BLOCK "Cascade_start_timer"   // DB42
{ S7_Optimized_Access := 'TRUE' }
AUTHOR : Simatic
FAMILY : IEC
NAME : IEC_TMR
VERSION : 1.0
// stored: InstanceOfName IEC_TIMER
"IEC_TIMER"
BEGIN
END_DATA_BLOCK

DATA_BLOCK "IEC_Timer_0_DB"   // DB50
{ S7_Optimized_Access := 'TRUE' }
AUTHOR : Simatic
FAMILY : IEC
NAME : IEC_TMR
VERSION : 1.0
// stored: InstanceOfName IEC_TIMER
"IEC_TIMER"
BEGIN
END_DATA_BLOCK

// folder: (top level)

FUNCTION_BLOCK "DI_Single"   // FB1, LAD
{ S7_Optimized_Access := 'TRUE' }
VERSION : 0.1
   VAR_INPUT
      input : Bool;
      delay_time : Time;
      filter : Bool;
      reverse : Bool;
   END_VAR
   VAR_OUTPUT
      value : Bool;
   END_VAR
   VAR
      TON : IEC_TIMER;
      TOF : IEC_TIMER;
   END_VAR
   VAR_TEMP   // added for the SCL form of the ladder/FBD networks
      _w1 : Bool;
      _w2 : Bool;
   END_VAR
BEGIN

REGION Network 1
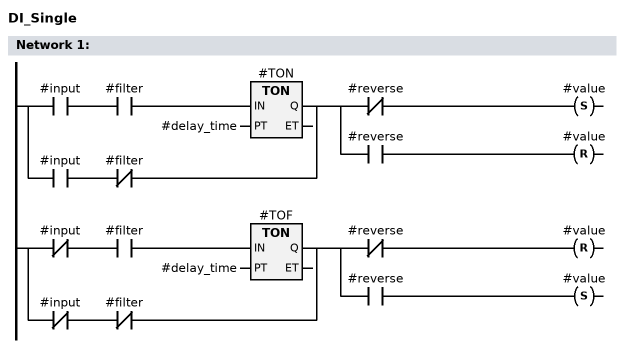
   #TON.TON(IN := #input AND #filter, PT := #delay_time);
   #_w1 := #TON.Q OR (#input AND NOT #filter);
   IF #_w1 AND NOT #reverse THEN #value := TRUE; END_IF;
   IF #_w1 AND #reverse THEN #value := FALSE; END_IF;
   #TOF.TON(IN := NOT #input AND #filter, PT := #delay_time);
   #_w2 := #TOF.Q OR (NOT #input AND NOT #filter);
   IF #_w2 AND NOT #reverse THEN #value := FALSE; END_IF;
   IF #_w2 AND #reverse THEN #value := TRUE; END_IF;
END_REGION
END_FUNCTION_BLOCK

FUNCTION_BLOCK "Gate_Valve_Error"   // FB2, LAD
{ S7_Optimized_Access := 'TRUE' }
VERSION : 0.1
   VAR_INPUT
      ChannelOpenOFF : Bool;
      ChannelCloseOFF : Bool;
      SignalOpen : Bool;
      SignalClose : Bool;
      ErrorOpen : Bool;
      ErrorClose : Bool;
   END_VAR
   VAR_OUTPUT
      ERROR : Bool;
   END_VAR
   VAR
      TON : IEC_TIMER;
   END_VAR
BEGIN

REGION Network 1
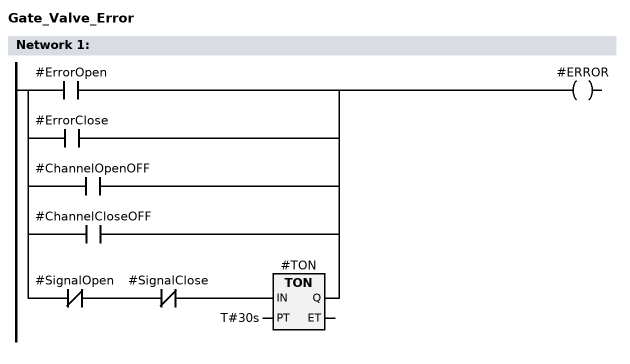
   #TON.TON(IN := NOT #SignalOpen AND NOT #SignalClose, PT := T#30s);
   #ERROR := #ErrorOpen OR #ErrorClose OR #ChannelOpenOFF OR #ChannelCloseOFF OR #TON.Q;
END_REGION
END_FUNCTION_BLOCK

FUNCTION_BLOCK "AI_Redundancy"   // FB3, SCL
{ S7_Optimized_Access := 'TRUE' }
VERSION : 0.1
   VAR_INPUT
      IN_AI_01 : Real;   // Сигнал 01
      IN_AI_02 : Real;   // Сигнал 02
      IN_Err_Proc : Real;   // Предельная разность сигналов
   END_VAR
   VAR_OUTPUT
      OUT_Error : Bool;   // Сигналы различаются больше чем на IN_Err_Proc %
      OUT_Result : Real;   // Результатирующий сигнал
   END_VAR
   VAR
      Error_1 : Real;
      Error_2 : Real;
   END_VAR
BEGIN
   #Error_1 := ABS(#IN_AI_01 - #IN_AI_02)*100.0 / #IN_AI_02;
   #Error_2 := ABS(#IN_AI_01 - #IN_AI_02)*100.0/ #IN_AI_01;
   IF #Error_1 > #IN_Err_Proc OR #Error_2 > #IN_Err_Proc THEN
       #OUT_Error := TRUE;
   ELSE
       #OUT_Error := FALSE;
   END_IF;

   IF #OUT_Error THEN
       #OUT_Result := MAX(IN1 := #IN_AI_01, IN2 := #IN_AI_02);
   ELSE
       #OUT_Result := (#IN_AI_01 + #IN_AI_02) / 2;
   END_IF;
END_FUNCTION_BLOCK

FUNCTION_BLOCK "Pump_Error"   // FB5, LAD
{ S7_Optimized_Access := 'TRUE' }
VERSION : 0.1
   VAR_INPUT
      DQ : Bool;
      STATE_Switch : Bool;
      STATE_Starter : Bool;
      SENSOR_Ball_Valve : Bool;
      SENSOR_High_Pressure_Pump : Real;
      SENSOR_High_Pressure_Pump_Error : Bool;
      Error_no_water : Bool;
   END_VAR
   VAR_OUTPUT
      Error : Bool;
   END_VAR
   VAR
      TP : IEC_TIMER;
      TON_1 : IEC_TIMER;
      TON_2 : IEC_TIMER;
      Error_1 : Bool;
      Error_2 : Bool;
   END_VAR
BEGIN

REGION Network 1
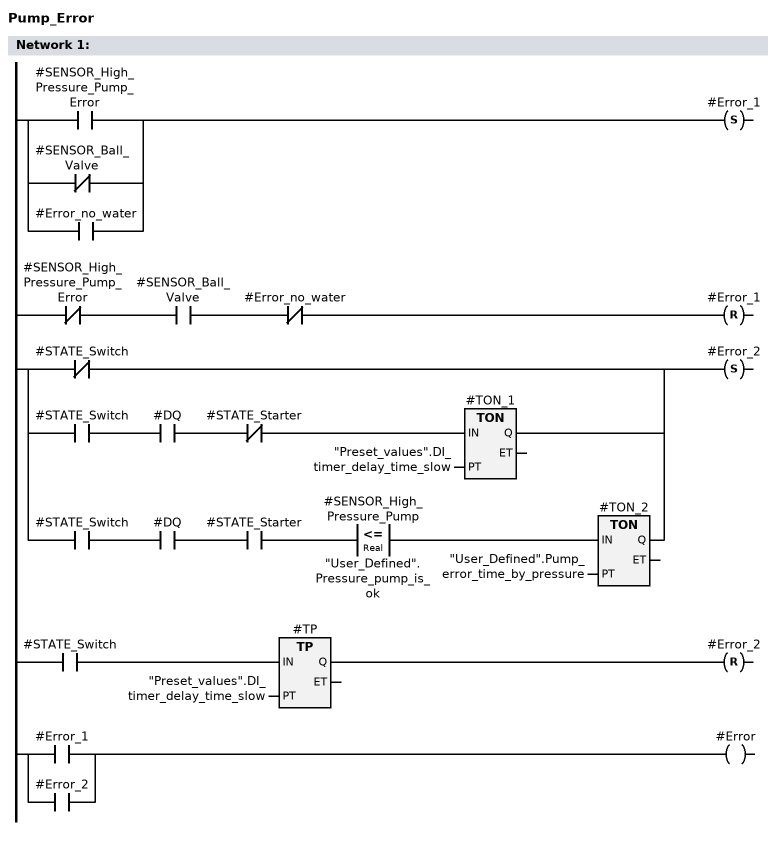
   IF #SENSOR_High_Pressure_Pump_Error OR NOT #SENSOR_Ball_Valve OR #Error_no_water THEN
       #Error_1 := TRUE;
   END_IF;
   IF NOT #SENSOR_High_Pressure_Pump_Error AND #SENSOR_Ball_Valve AND NOT #Error_no_water THEN
       #Error_1 := FALSE;
   END_IF;
   #TON_1.TON(IN := #STATE_Switch AND #DQ AND NOT #STATE_Starter,
              PT := "Preset_values".DI_timer_delay_time_slow);
   #TON_2.TON(IN := #STATE_Switch AND #DQ AND #STATE_Starter AND (#SENSOR_High_Pressure_Pump <= "User_Defined".Pressure_pump_is_ok),
              PT := "User_Defined".Pump_error_time_by_pressure);
   IF NOT #STATE_Switch OR #TON_1.Q OR #TON_2.Q THEN #Error_2 := TRUE; END_IF;
   #TP.TP(IN := #STATE_Switch, PT := "Preset_values".DI_timer_delay_time_slow);
   IF #TP.Q THEN #Error_2 := FALSE; END_IF;
   #Error := #Error_1 OR #Error_2;
END_REGION
END_FUNCTION_BLOCK

FUNCTION_BLOCK "First_pump_start"   // FB6, SCL
{ S7_Optimized_Access := 'TRUE' }
VERSION : 0.1
   VAR_INPUT
      Total_pumps : Int;
      Signal_Fire : Bool;
      StatePumpWork : Array[1..10] of Bool;
      PumpError : Array[1..10] of Bool;
   END_VAR
   VAR_IN_OUT
      First_Pump_has_started : Bool;
      PumpRun : Array[1..10] of Bool;
   END_VAR
   VAR
      init : Bool := true;
   END_VAR
   VAR_TEMP
      "Counter" : Int;
      Start_pump : Bool;
   END_VAR
BEGIN
   IF #init OR NOT #Signal_Fire THEN
       #First_Pump_has_started := false;
       #init := false;
   END_IF;

   IF #Signal_Fire
       AND NOT #First_Pump_has_started
   THEN
       FOR #Counter := 1 TO #Total_pumps DO
           IF NOT #PumpError[#Counter]
               AND NOT #StatePumpWork[#Counter]
           THEN
               #PumpRun[#Counter] := TRUE;
               #First_Pump_has_started := TRUE;
               EXIT;
           END_IF;
       END_FOR;
   END_IF;
END_FUNCTION_BLOCK

FUNCTION_BLOCK "State_work_pump"   // FB7, SCL
{ S7_Optimized_Access := 'TRUE' }
VERSION : 0.1
   VAR_INPUT
      Total_pumps : SInt;
   END_VAR
   VAR_TEMP
      "Counter" : SInt;
   END_VAR
BEGIN
   FOR #Counter := 1 TO #Total_pumps DO
       IF "Pumps_data".State_switch_pump[#Counter] AND "Pumps_data".State_starter_pump[#Counter] THEN
           "Pumps_data".State_work_pump[#Counter] := TRUE;
           ;
       ELSE
           "Pumps_data".State_work_pump[#Counter] := FALSE;
           ;
       END_IF;
   END_FOR;
   CASE #Total_pumps OF
       1:
           IF "Pumps_data".State_work_pump[1] THEN
               "Pumps_data".State_work_any_pump := TRUE;
           ELSE
               "Pumps_data".State_work_any_pump := FALSE;
           END_IF;
           ;
       2:
           IF "Pumps_data".State_work_pump[1] OR
               "Pumps_data".State_work_pump[2] THEN
               "Pumps_data".State_work_any_pump := TRUE;
           ELSE
               "Pumps_data".State_work_any_pump := FALSE;
           END_IF;
           ;
       3:
           IF "Pumps_data".State_work_pump[1] OR
               "Pumps_data".State_work_pump[2] OR
               "Pumps_data".State_work_pump[3] THEN
               "Pumps_data".State_work_any_pump := TRUE;
           ELSE
               "Pumps_data".State_work_any_pump := FALSE;
           END_IF;
           ;
       4:
           IF "Pumps_data".State_work_pump[1] OR
               "Pumps_data".State_work_pump[2] OR
               "Pumps_data".State_work_pump[3] OR
               "Pumps_data".State_work_pump[4] THEN
               "Pumps_data".State_work_any_pump := TRUE;
           ELSE
               "Pumps_data".State_work_any_pump := FALSE;
           END_IF;
           ;
       5:
           IF "Pumps_data".State_work_pump[1] OR
               "Pumps_data".State_work_pump[2] OR
               "Pumps_data".State_work_pump[3] OR
               "Pumps_data".State_work_pump[4] OR
               "Pumps_data".State_work_pump[5] THEN
               "Pumps_data".State_work_any_pump := TRUE;
           ELSE
               "Pumps_data".State_work_any_pump := FALSE;
           END_IF;
           ;
       6:
           IF "Pumps_data".State_work_pump[1] OR
               "Pumps_data".State_work_pump[2] OR
               "Pumps_data".State_work_pump[3] OR
               "Pumps_data".State_work_pump[4] OR
               "Pumps_data".State_work_pump[5] OR
               "Pumps_data".State_work_pump[6] THEN
               "Pumps_data".State_work_any_pump := TRUE;
           ELSE
               "Pumps_data".State_work_any_pump := FALSE;
           END_IF;
           ;
       7:
           IF "Pumps_data".State_work_pump[1] OR
               "Pumps_data".State_work_pump[2] OR
               "Pumps_data".State_work_pump[3] OR
               "Pumps_data".State_work_pump[4] OR
               "Pumps_data".State_work_pump[5] OR
               "Pumps_data".State_work_pump[6] OR
               "Pumps_data".State_work_pump[7] THEN
               "Pumps_data".State_work_any_pump := TRUE;
           ELSE
               "Pumps_data".State_work_any_pump := FALSE;
           END_IF;
           ;
       8:
           IF "Pumps_data".State_work_pump[1] OR
               "Pumps_data".State_work_pump[2] OR
               "Pumps_data".State_work_pump[3] OR
               "Pumps_data".State_work_pump[4] OR
               "Pumps_data".State_work_pump[5] OR
               "Pumps_data".State_work_pump[6] OR
               "Pumps_data".State_work_pump[7] OR
               "Pumps_data".State_work_pump[8] THEN
               "Pumps_data".State_work_any_pump := TRUE;
           ELSE
               "Pumps_data".State_work_any_pump := FALSE;
           END_IF;
           ;
       9:
           IF "Pumps_data".State_work_pump[1] OR
               "Pumps_data".State_work_pump[2] OR
               "Pumps_data".State_work_pump[3] OR
               "Pumps_data".State_work_pump[4] OR
               "Pumps_data".State_work_pump[5] OR
               "Pumps_data".State_work_pump[6] OR
               "Pumps_data".State_work_pump[7] OR
               "Pumps_data".State_work_pump[8] OR
               "Pumps_data".State_work_pump[9] THEN
               "Pumps_data".State_work_any_pump := TRUE;
           ELSE
               "Pumps_data".State_work_any_pump := FALSE;
           END_IF;
           ;
       10:
           IF "Pumps_data".State_work_pump[1] OR
               "Pumps_data".State_work_pump[2] OR
               "Pumps_data".State_work_pump[3] OR
               "Pumps_data".State_work_pump[4] OR
               "Pumps_data".State_work_pump[5] OR
               "Pumps_data".State_work_pump[6] OR
               "Pumps_data".State_work_pump[7] OR
               "Pumps_data".State_work_pump[8] OR
               "Pumps_data".State_work_pump[9] OR
               "Pumps_data".State_work_pump[10] THEN
               "Pumps_data".State_work_any_pump := TRUE;
           ELSE
               "Pumps_data".State_work_any_pump := FALSE;
           END_IF;
           ;
   END_CASE;
END_FUNCTION_BLOCK

FUNCTION_BLOCK "Sound_PTO"   // FB8, LAD
{ S7_Optimized_Access := 'TRUE' }
VERSION : 0.1
   VAR_INPUT
      Hardware_ID : Hw_Pto;
      Button_sound_off : Bool;
      ERROR_any : Bool;
      SIGNAL_fire : Bool;
      STATE_work_any_pump : Bool;
      Error_frequency : UDInt := 1;
      Fire_frequency : UDInt := 2;
      Work_frequency : UDInt := 50;
   END_VAR
   VAR_OUTPUT
      Led_sound_off : Bool;
   END_VAR
   VAR
      Frequency : UDInt;
      Sound_off : Bool;
   END_VAR
   VAR_TEMP   // added for the SCL form of the ladder/FBD networks
      _w1 : Bool;
      _w2 : Bool;
   END_VAR
BEGIN

REGION Network 1
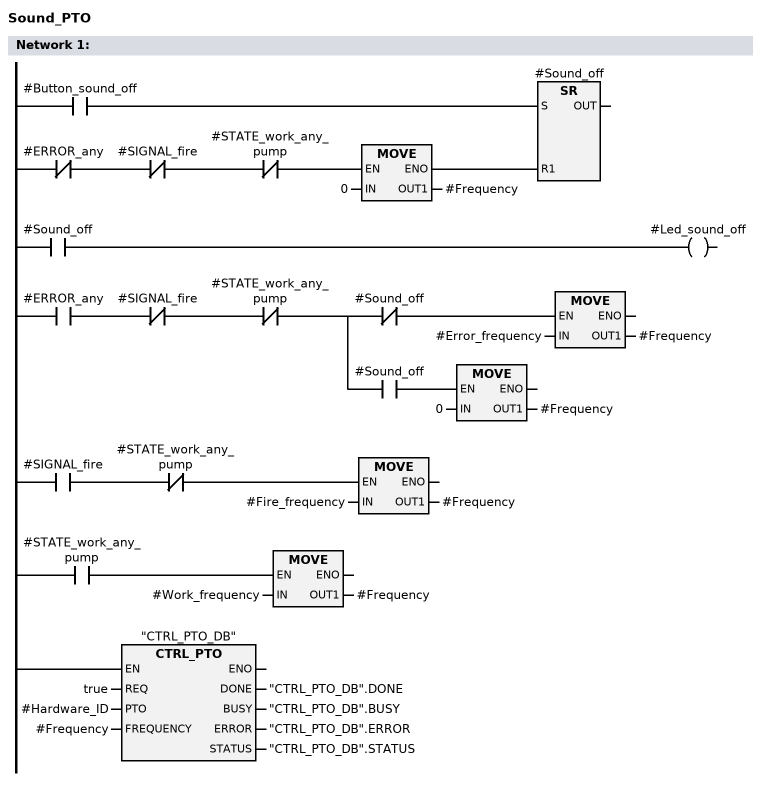
   #_w1 := NOT #ERROR_any AND NOT #SIGNAL_fire AND NOT #STATE_work_any_pump;
   IF #_w1 THEN #Frequency := 0; END_IF;
   IF #Button_sound_off THEN
       #Sound_off := TRUE;   // SR flip-flop
   END_IF;
   IF #_w1 THEN #Sound_off := FALSE; END_IF;
   #Led_sound_off := #Sound_off;
   #_w2 := #ERROR_any AND NOT #SIGNAL_fire AND NOT #STATE_work_any_pump;
   IF #_w2 AND NOT #Sound_off THEN #Frequency := #Error_frequency; END_IF;
   IF #_w2 AND #Sound_off THEN #Frequency := 0; END_IF;
   IF #SIGNAL_fire AND NOT #STATE_work_any_pump THEN #Frequency := #Fire_frequency; END_IF;
   IF #STATE_work_any_pump THEN #Frequency := #Work_frequency; END_IF;
   "CTRL_PTO_DB"(REQ := true,   // CTRL_PTO
                 PTO := #Hardware_ID,
                 FREQUENCY := #Frequency,
                 DONE => "CTRL_PTO_DB".DONE,
                 BUSY => "CTRL_PTO_DB".BUSY,
                 ERROR => "CTRL_PTO_DB".ERROR,
                 STATUS => "CTRL_PTO_DB".STATUS);
END_REGION
END_FUNCTION_BLOCK

FUNCTION_BLOCK "SOVA_Modbus_Input_Reading"   // FB9, SCL
{ S7_Optimized_Access := 'TRUE' }
VERSION : 0.1
   VAR_INPUT
      Device_total : Int;
      Port : Hw_SubModule;
   END_VAR
   VAR_TEMP
      "Counter" : Int;
      Master_reading_done : Bool;
      Sova_input_counter : Int;
      COMM_LOAD_DONE : Bool;
   END_VAR
BEGIN
   "MB_COMM_LOAD_DB"(REQ:="FirstScan",
                     "PORT":=#Port,
                     BAUD:=9600,
                     DONE=>#COMM_LOAD_DONE,
                     MB_DB:="MB_MASTER_DB");

   IF #COMM_LOAD_DONE THEN
       FOR #Counter := 1 TO #Device_total DO
           #Master_reading_done := FALSE;
           "MB_MASTER_DB"(REQ := TRUE,
                          MB_ADDR := #Counter,
                          MODE := 0,
                          DATA_ADDR := 40003,
                          DONE => #Master_reading_done,
                          DATA_LEN := 12,
                          DATA_PTR := "SOVA_Modbus_Input".SOVA[#Counter]);
           IF #Master_reading_done = TRUE THEN
               #Master_reading_done := FALSE;
               FOR #Sova_input_counter := 1 TO 12 DO




                   CASE "SOVA_Modbus_Input".SOVA[#Counter,#Sova_input_counter] OF
                       0: // Channel off - SOVA
                           "SOVA_Modbus_Input".MB_Line[#Counter, #Sova_input_counter, 0] := true;
                           "SOVA_Modbus_Input".MB_Line[#Counter, #Sova_input_counter, 7] := true;//error variable

                           "SOVA_Modbus_Input".MB_Line[#Counter, #Sova_input_counter, 1] := FALSE;
                           "SOVA_Modbus_Input".MB_Line[#Counter, #Sova_input_counter, 2] := FALSE;
                           "SOVA_Modbus_Input".MB_Line[#Counter, #Sova_input_counter, 3] := FALSE;
                           "SOVA_Modbus_Input".MB_Line[#Counter, #Sova_input_counter, 4] := FALSE;
                           "SOVA_Modbus_Input".MB_Line[#Counter, #Sova_input_counter, 5] := FALSE;
                           "SOVA_Modbus_Input".MB_Line[#Counter, #Sova_input_counter, 6] := FALSE;
                           ;
                       1: // Channel on - SOVA

                           "SOVA_Modbus_Input".MB_Line[#Counter, #Sova_input_counter, 1] := true;
                           "SOVA_Modbus_Input".MB_Line[#Counter, #Sova_input_counter, 0] := FALSE;
                           "SOVA_Modbus_Input".MB_Line[#Counter, #Sova_input_counter, 2] := FALSE;
                           "SOVA_Modbus_Input".MB_Line[#Counter, #Sova_input_counter, 3] := FALSE;
                           "SOVA_Modbus_Input".MB_Line[#Counter, #Sova_input_counter, 4] := FALSE;
                           "SOVA_Modbus_Input".MB_Line[#Counter, #Sova_input_counter, 5] := FALSE;
                           "SOVA_Modbus_Input".MB_Line[#Counter, #Sova_input_counter, 6] := FALSE;
                           "SOVA_Modbus_Input".MB_Line[#Counter, #Sova_input_counter, 7] := FALSE;
                       2: // Signal1 - SOVA

                           "SOVA_Modbus_Input".MB_Line[#Counter, #Sova_input_counter, 2] := true;
                           "SOVA_Modbus_Input".MB_Line[#Counter, #Sova_input_counter, 6] := true; //signal variable

                           "SOVA_Modbus_Input".MB_Line[#Counter, #Sova_input_counter, 0] := FALSE;
                           "SOVA_Modbus_Input".MB_Line[#Counter, #Sova_input_counter, 1] := FALSE;
                           "SOVA_Modbus_Input".MB_Line[#Counter, #Sova_input_counter, 3] := FALSE;
                           "SOVA_Modbus_Input".MB_Line[#Counter, #Sova_input_counter, 4] := FALSE;
                           "SOVA_Modbus_Input".MB_Line[#Counter, #Sova_input_counter, 5] := FALSE;
                           "SOVA_Modbus_Input".MB_Line[#Counter, #Sova_input_counter, 7] := FALSE;

                       3: // Signal2 - SOVA
                           "SOVA_Modbus_Input".MB_Line[#Counter, #Sova_input_counter, 3] := true;
                           "SOVA_Modbus_Input".MB_Line[#Counter, #Sova_input_counter, 6] := true; //signal variable

                           "SOVA_Modbus_Input".MB_Line[#Counter, #Sova_input_counter, 0] := FALSE;
                           "SOVA_Modbus_Input".MB_Line[#Counter, #Sova_input_counter, 1] := FALSE;
                           "SOVA_Modbus_Input".MB_Line[#Counter, #Sova_input_counter, 2] := FALSE;
                           "SOVA_Modbus_Input".MB_Line[#Counter, #Sova_input_counter, 4] := FALSE;
                           "SOVA_Modbus_Input".MB_Line[#Counter, #Sova_input_counter, 5] := FALSE;
                           "SOVA_Modbus_Input".MB_Line[#Counter, #Sova_input_counter, 7] := FALSE;
                       4: // Wire broken - SOVA
                           "SOVA_Modbus_Input".MB_Line[#Counter, #Sova_input_counter, 4] := true;
                           "SOVA_Modbus_Input".MB_Line[#Counter, #Sova_input_counter, 7] := true; //error variable

                           "SOVA_Modbus_Input".MB_Line[#Counter, #Sova_input_counter, 0] := FALSE;
                           "SOVA_Modbus_Input".MB_Line[#Counter, #Sova_input_counter, 1] := FALSE;
                           "SOVA_Modbus_Input".MB_Line[#Counter, #Sova_input_counter, 2] := FALSE;
                           "SOVA_Modbus_Input".MB_Line[#Counter, #Sova_input_counter, 3] := FALSE;
                           "SOVA_Modbus_Input".MB_Line[#Counter, #Sova_input_counter, 5] := FALSE;
                           "SOVA_Modbus_Input".MB_Line[#Counter, #Sova_input_counter, 6] := FALSE;
                       5: // Circuit Short - SOVA
                           "SOVA_Modbus_Input".MB_Line[#Counter, #Sova_input_counter, 5] := true;
                           "SOVA_Modbus_Input".MB_Line[#Counter, #Sova_input_counter, 7] := true; //error variable

                           "SOVA_Modbus_Input".MB_Line[#Counter, #Sova_input_counter, 0] := FALSE;
                           "SOVA_Modbus_Input".MB_Line[#Counter, #Sova_input_counter, 1] := FALSE;
                           "SOVA_Modbus_Input".MB_Line[#Counter, #Sova_input_counter, 2] := FALSE;
                           "SOVA_Modbus_Input".MB_Line[#Counter, #Sova_input_counter, 3] := FALSE;
                           "SOVA_Modbus_Input".MB_Line[#Counter, #Sova_input_counter, 4] := FALSE;
                           "SOVA_Modbus_Input".MB_Line[#Counter, #Sova_input_counter, 6] := FALSE;

                   END_CASE;

               END_FOR;

           END_IF;
       END_FOR;
   END_IF;
END_FUNCTION_BLOCK

FUNCTION_BLOCK "Standby_Pump/Compressor_Error"   // FB10, LAD
{ S7_Optimized_Access := 'TRUE' }
VERSION : 0.1
   VAR_INPUT
      DQ : Bool;
      STATE_Switch : Bool;
      STATE_Starter : Bool;
      ERROR_no_water : Bool;
   END_VAR
   VAR_OUTPUT
      Error : Bool;
   END_VAR
   VAR
      TP : IEC_TIMER;
      TON : IEC_TIMER;
   END_VAR
BEGIN

REGION Network 1
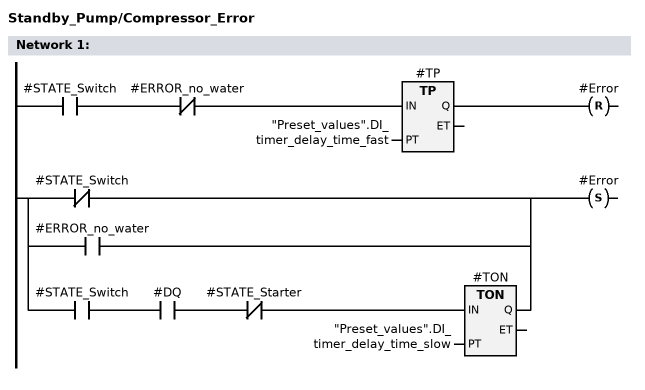
   #TP.TP(IN := #STATE_Switch AND NOT #ERROR_no_water, PT := "Preset_values".DI_timer_delay_time_fast);
   IF #TP.Q THEN #Error := FALSE; END_IF;
   #TON.TON(IN := #STATE_Switch AND #DQ AND NOT #STATE_Starter, PT := "Preset_values".DI_timer_delay_time_slow);
   IF NOT #STATE_Switch OR #ERROR_no_water OR #TON.Q THEN #Error := TRUE; END_IF;
END_REGION
END_FUNCTION_BLOCK

FUNCTION_BLOCK "AI_Sensor"   // FB11, LAD
{ S7_Optimized_Access := 'TRUE' }
VERSION : 0.1
   VAR_INPUT
      In : Int;
      Int_HL : Int := 27468;
      Int_LL : Int := 0;
      Value_HL : Real;
      Value_LL : Real;
   END_VAR
   VAR_OUTPUT
      Value : Real;
      Error : Bool;
   END_VAR
   VAR_TEMP
      In_real : Real;
   END_VAR
BEGIN

REGION Network 1
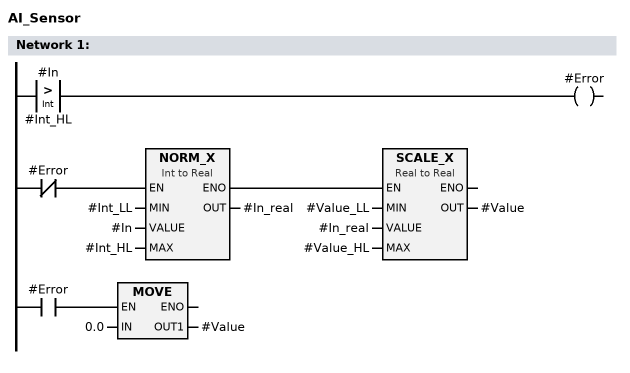
   RUNG wire#powerrail
      { S7_Templates := "SrcType := Int" } GT_Contact(in1 := #In, in2 := #Int_HL)
      Coil( #Error )
   END_RUNG
   RUNG wire#powerrail
      I_Contact( #Error )
      { S7_Templates := "[SrcType := Int, DestType := Real]" } Normalize(min := #Int_LL, value := #In, max := #Int_HL, out => #In_real)
      { S7_Templates := "[SrcType := Real, DestType := Real]" } Scale(min := #Value_LL, value := #In_real, max := #Value_HL, out => #Value)
   END_RUNG
   RUNG wire#powerrail
      Contact( #Error )
      Move(in := 0.0, out1 => #Value)
   END_RUNG
   // the same network as SCL:
   #Error := #In > #Int_HL;
   IF NOT #Error THEN
       #In_real := NORM_X(MIN := #Int_LL, VALUE := #In, MAX := #Int_HL);
       #Value := SCALE_X(MIN := #Value_LL, VALUE := #In_real, MAX := #Value_HL);
   END_IF;
   IF #Error THEN #Value := 0.0; END_IF;
END_REGION
END_FUNCTION_BLOCK

FUNCTION_BLOCK "ModbusMasterConnector"   // FB12, SCL
{ S7_Optimized_Access := 'FALSE' }
VERSION : 0.1
   VAR_INPUT
      PORT : Hw_SubModule;
   END_VAR
   VAR
      instModbusCommLoad : Modbus_Comm_Load;
      instModbusMaster : Modbus_Master;
      init : Bool := True;
      BAUD : UDInt := 9600;
      STOP_BITS : USInt := 1;
      PARITY : UInt;
      Read_REGS : Word;
      "Step" : UInt;
      Write_REGS : Array[0..38] of Word;
   END_VAR
BEGIN
   IF #init THEN
       #Step := 2;
       #instModbusCommLoad.MODE := 4;
       #instModbusCommLoad.STOP_BITS := #STOP_BITS;
   END_IF;

   #instModbusCommLoad(REQ := #init,
                       "PORT" := #PORT,
                       BAUD := #BAUD,
                       PARITY := #PARITY,
                       MB_DB := #instModbusMaster.MB_DB);

   #init := FALSE;

   CASE #Step OF
       1:

           #instModbusMaster(REQ := TRUE,
                             MB_ADDR := 1,
                             MODE := 0,
                             DATA_ADDR := 40001,
                             DATA_LEN := 1,
                             DATA_PTR := #Read_REGS);
           IF #instModbusMaster.DONE THEN
               #Step := 2;
               "ReadHoldingRegister" := #Read_REGS;
               //Maping  registers
               #Write_REGS[0]:= "WriteHoldingRegister_00";
               #Write_REGS[1] := "WriteHoldingRegister_01";
               #Write_REGS[2] := "WriteHoldingRegister_02";
               #Write_REGS[3] := "WriteHoldingRegister_03";
               #Write_REGS[4] := "WriteHoldingRegister_04";
               #Write_REGS[5] := "WriteHoldingRegister_05";
               #Write_REGS[6] := "WriteHoldingRegister_06";
               #Write_REGS[7] := "WriteHoldingRegister_07";
               #Write_REGS[8] := "WriteHoldingRegister_08";
               #Write_REGS[9] := "WriteHoldingRegister_09";
               #Write_REGS[10] := "WriteHoldingRegister_10";
               #Write_REGS[11] := "WriteHoldingRegister_11";
               #Write_REGS[12] := "WriteHoldingRegister_12";
               #Write_REGS[13] := "WriteHoldingRegister_13";
               #Write_REGS[14] := "WriteHoldingRegister_14";
               #Write_REGS[15] := "WriteHoldingRegister_15";
               #Write_REGS[16] := "WriteHoldingRegister_16";
               #Write_REGS[17] := "WriteHoldingRegister_17";
               #Write_REGS[18] := "WriteHoldingRegister_18";
               #Write_REGS[19] := "WriteHoldingRegister_19";
               #Write_REGS[20] := "WriteHoldingRegister_20";
               #Write_REGS[21] := "WriteHoldingRegister_21";
               #Write_REGS[22] := "WriteHoldingRegister_22";
               #Write_REGS[23] := "WriteHoldingRegister_23";
               #Write_REGS[24] := "WriteHoldingRegister_24";
               #Write_REGS[25] := "WriteHoldingRegister_25";
               #Write_REGS[26] := "WriteHoldingRegister_26";
               #Write_REGS[27] := "WriteHoldingRegister_27";
               #Write_REGS[28] := "WriteHoldingRegister_28";
               #Write_REGS[29] := "WriteHoldingRegister_29";
               #Write_REGS[30] := "WriteHoldingRegister_30";
               #Write_REGS[31] := "WriteHoldingRegister_31";
               #Write_REGS[32] := "WriteHoldingRegister_32";
               #Write_REGS[33] := "WriteHoldingRegister_33";
               #Write_REGS[34] := "WriteHoldingRegister_34";
               #Write_REGS[35] := "WriteHoldingRegister_35";
               #Write_REGS[36] := "WriteHoldingRegister_36";
               #Write_REGS[37] := "WriteHoldingRegister_37";
               #Write_REGS[38] := "WriteHoldingRegister_38";



           END_IF;

           IF #instModbusMaster.ERROR THEN
               #Step := 2;
           END_IF;
       2:
           #instModbusMaster(REQ := TRUE,
                             MB_ADDR := 1,
                             MODE := 1,
                             DATA_ADDR := 40002,
                             DATA_LEN := 39,
                             DATA_PTR := #Write_REGS);
           IF #instModbusMaster.DONE THEN
               #Step := 1;


           END_IF;
           IF #instModbusMaster.ERROR THEN
               #Step := 1;
           END_IF;
   END_CASE;
END_FUNCTION_BLOCK

FUNCTION_BLOCK "Cascade"   // FB13, SCL
{ S7_Optimized_Access := 'TRUE' }
VERSION : 0.1
   VAR_INPUT
      CascadeStart : Real := 0.0;
      CascadeStop : Real;
      TotalPumps : Int;
      PumpError : Array[1..10] of Bool;
      PumpWorkState : Array[1..10] of Bool;
      FirstPumpHasStarted : Bool;
      PressureGlobal : Real;
   END_VAR
   VAR_IN_OUT
      PumpRun : Array[1..10] of Bool;
   END_VAR
   VAR_TEMP
      CounterStart : Int;
      CounterStop : Int;
   END_VAR
BEGIN
   IF #FirstPumpHasStarted AND #PressureGlobal < #CascadeStart AND "Pumps_data".Error_any_pump THEN
       FOR #CounterStart := 1 TO #TotalPumps DO
               IF NOT #PumpError[#CounterStart] AND NOT #PumpWorkState[#CounterStart] THEN
                   #PumpRun[#CounterStart] := TRUE;
                   EXIT;
               END_IF;
        END_FOR;
   ELSIF #FirstPumpHasStarted AND #PressureGlobal < #CascadeStart AND NOT "Pumps_data".Error_any_pump THEN
        FOR #CounterStart := 1 TO #TotalPumps - 1 DO
               IF NOT #PumpError[#CounterStart] AND NOT #PumpWorkState[#CounterStart] THEN
                   #PumpRun[#CounterStart] := TRUE;
                   EXIT;
               END_IF;
        END_FOR;
   END_IF;
   IF #FirstPumpHasStarted AND #PressureGlobal > #CascadeStop AND "Pumps_data".pump_work_counter > 1 THEN
       FOR #CounterStop := #TotalPumps TO 1 BY -1 DO
           IF NOT #PumpError[#CounterStop] AND #PumpWorkState[#CounterStop] THEN
               #PumpRun[#CounterStop] := FALSE;
               EXIT;
           END_IF;
       END_FOR;
   END_IF;
END_FUNCTION_BLOCK

FUNCTION_BLOCK "PumpRun"   // FB14, LAD
{ S7_Optimized_Access := 'TRUE' }
VERSION : 0.1
   VAR_INPUT
      Error : Bool;
      ModeAuto : Bool;
      ButtonStop : Bool;
      KPPUButtonStop : Bool;
      FirstPumpHasStarted : Bool;
      PumpRunCommand : Bool;
      CascadeTimer : Time;
      Pressure : Real;
   END_VAR
   VAR_OUTPUT
      DQ : Bool;
   END_VAR
   VAR
      TON : IEC_TIMER;
      TOF : IEC_TIMER;
      TON_2 : IEC_TIMER;
   END_VAR
BEGIN

REGION Network 1
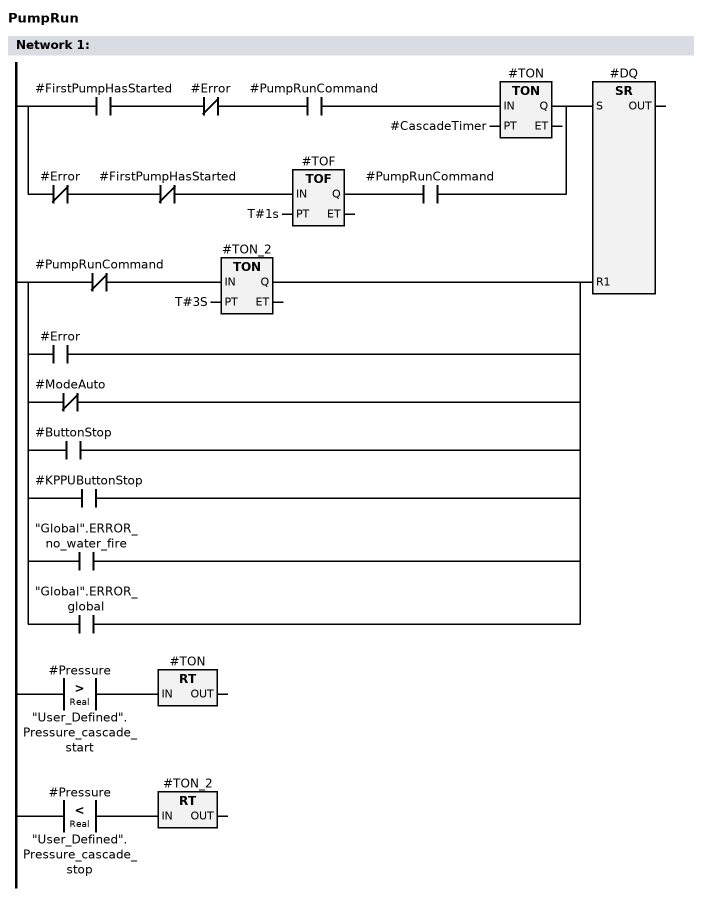
   #TON.TON(IN := #FirstPumpHasStarted AND NOT #Error AND #PumpRunCommand, PT := #CascadeTimer);
   #TOF.TOF(IN := NOT #Error AND NOT #FirstPumpHasStarted, PT := T#1s);
   #TON_2.TON(IN := NOT #PumpRunCommand, PT := T#3S);
   IF #TON.Q OR (#TOF.Q AND #PumpRunCommand) THEN
       #DQ := TRUE;   // SR flip-flop
   END_IF;
   IF #TON_2.Q OR #Error OR NOT #ModeAuto OR #ButtonStop OR #KPPUButtonStop OR "Global".ERROR_no_water_fire OR "Global".ERROR_global THEN
       #DQ := FALSE;
   END_IF;
   IF #Pressure > "User_Defined".Pressure_cascade_start THEN RESET_TIMER(#TON); END_IF;
   IF #Pressure < "User_Defined".Pressure_cascade_stop THEN RESET_TIMER(#TON_2); END_IF;
END_REGION
END_FUNCTION_BLOCK

FUNCTION "DI_All" : Void   // FC1, LAD
{ S7_Optimized_Access := 'TRUE' }
VERSION : 0.1
   VAR_TEMP   // added for the SCL form of the ladder/FBD networks
      _w1 : Bool;
      _w2 : Bool;
      _w3 : Bool;
      _w4 : Bool;
      _w5 : Bool;
      _w6 : Bool;
      _w7 : Bool;
      _w8 : Bool;
   END_VAR
BEGIN

REGION Network 1: Дискретные входы состояния ППУ
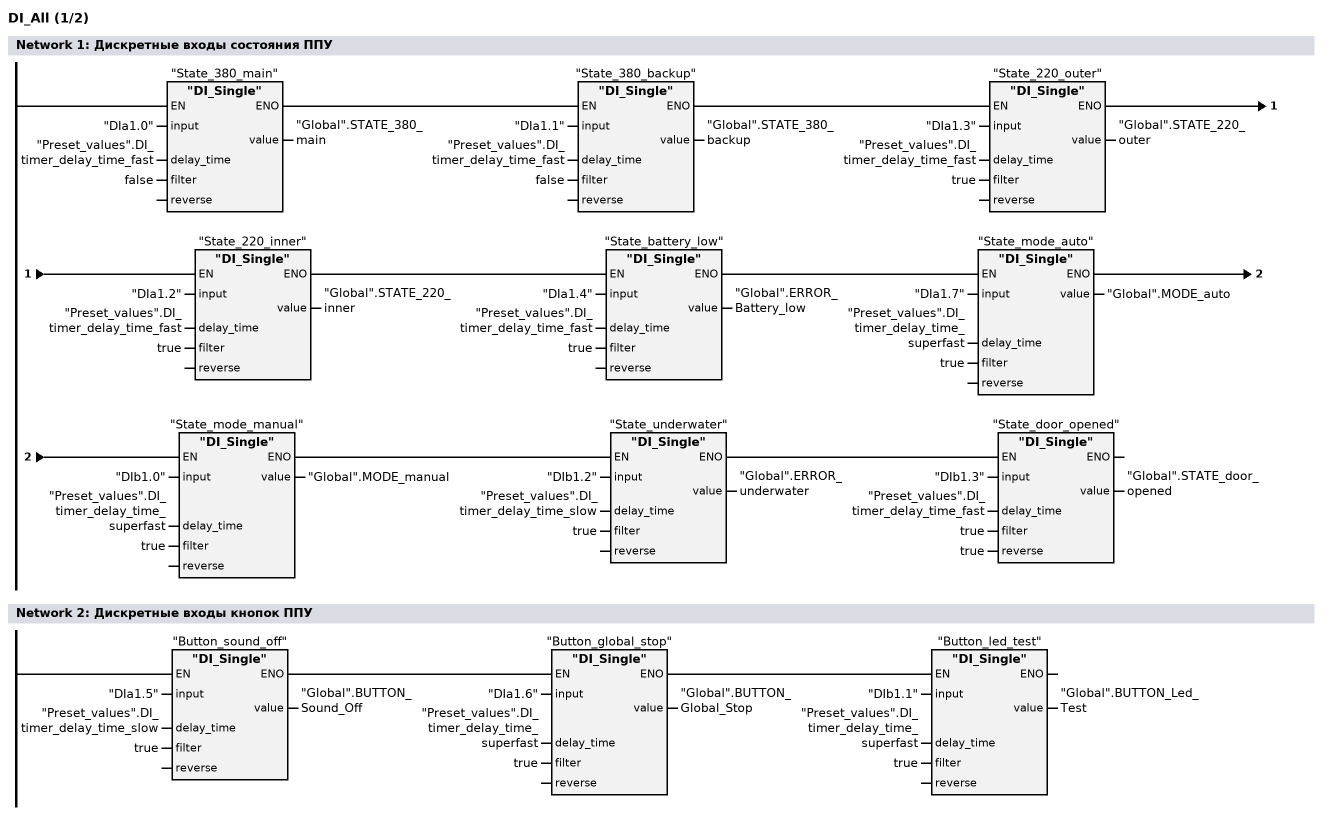
   RUNG wire#powerrail
      "State_380_main"(input := "DIa1.0", delay_time := "Preset_values".DI_timer_delay_time_fast, filter := false, reverse :=, value => "Global".STATE_380_main)
      "State_380_backup"(input := "DIa1.1", delay_time := "Preset_values".DI_timer_delay_time_fast, filter := false, reverse :=, value => "Global".STATE_380_backup)
      "State_220_outer"(input := "DIa1.3", delay_time := "Preset_values".DI_timer_delay_time_fast, filter := true, reverse :=, value => "Global".STATE_220_outer)
      "State_220_inner"(input := "DIa1.2", delay_time := "Preset_values".DI_timer_delay_time_fast, filter := true, reverse :=, value => "Global".STATE_220_inner)
      "State_battery_low"(input := "DIa1.4", delay_time := "Preset_values".DI_timer_delay_time_fast, filter := true, reverse :=, value => "Global".ERROR_Battery_low)
      "State_mode_auto"(input := "DIa1.7", delay_time := "Preset_values".DI_timer_delay_time_superfast, filter := true, reverse :=, value => "Global".MODE_auto)
      "State_mode_manual"(input := "DIb1.0", delay_time := "Preset_values".DI_timer_delay_time_superfast, filter := true, reverse :=, value => "Global".MODE_manual)
      "State_underwater"(input := "DIb1.2", delay_time := "Preset_values".DI_timer_delay_time_slow, filter := true, reverse :=, value => "Global".ERROR_underwater)
      "State_door_opened"(input := "DIb1.3", delay_time := "Preset_values".DI_timer_delay_time_fast, filter := true, reverse := true, value => "Global".STATE_door_opened)
   END_RUNG
   // the same network as SCL:
   "State_380_main"(input := "DIa1.0",   // "DI_Single"
                    delay_time := "Preset_values".DI_timer_delay_time_fast,
                    filter := false,
                    value => "Global".STATE_380_main,
                    ENO => #_w1);
   "State_380_backup"(EN := #_w1,   // "DI_Single"
                      input := "DIa1.1",
                      delay_time := "Preset_values".DI_timer_delay_time_fast,
                      filter := false,
                      value => "Global".STATE_380_backup,
                      ENO => #_w2);
   "State_220_outer"(EN := #_w2,   // "DI_Single"
                     input := "DIa1.3",
                     delay_time := "Preset_values".DI_timer_delay_time_fast,
                     filter := true,
                     value => "Global".STATE_220_outer,
                     ENO => #_w3);
   "State_220_inner"(EN := #_w3,   // "DI_Single"
                     input := "DIa1.2",
                     delay_time := "Preset_values".DI_timer_delay_time_fast,
                     filter := true,
                     value => "Global".STATE_220_inner,
                     ENO => #_w4);
   "State_battery_low"(EN := #_w4,   // "DI_Single"
                       input := "DIa1.4",
                       delay_time := "Preset_values".DI_timer_delay_time_fast,
                       filter := true,
                       value => "Global".ERROR_Battery_low,
                       ENO => #_w5);
   "State_mode_auto"(EN := #_w5,   // "DI_Single"
                     input := "DIa1.7",
                     delay_time := "Preset_values".DI_timer_delay_time_superfast,
                     filter := true,
                     value => "Global".MODE_auto,
                     ENO => #_w6);
   "State_mode_manual"(EN := #_w6,   // "DI_Single"
                       input := "DIb1.0",
                       delay_time := "Preset_values".DI_timer_delay_time_superfast,
                       filter := true,
                       value => "Global".MODE_manual,
                       ENO => #_w7);
   "State_underwater"(EN := #_w7,   // "DI_Single"
                      input := "DIb1.2",
                      delay_time := "Preset_values".DI_timer_delay_time_slow,
                      filter := true,
                      value => "Global".ERROR_underwater,
                      ENO => #_w8);
   IF #_w8 THEN
       "State_door_opened"(input := "DIb1.3",   // "DI_Single"
                           delay_time := "Preset_values".DI_timer_delay_time_fast,
                           filter := true,
                           reverse := true,
                           value => "Global".STATE_door_opened);
   END_IF;
END_REGION

REGION Network 2: Дискретные входы кнопок ППУ
   RUNG wire#powerrail
      "Button_sound_off"(input := "DIa1.5", delay_time := "Preset_values".DI_timer_delay_time_slow, filter := true, reverse :=, value => "Global".BUTTON_Sound_Off)
      "Button_global_stop"(input := "DIa1.6", delay_time := "Preset_values".DI_timer_delay_time_superfast, filter := true, reverse :=, value => "Global".BUTTON_Global_Stop)
      "Button_led_test"(input := "DIb1.1", delay_time := "Preset_values".DI_timer_delay_time_superfast, filter := true, reverse :=, value => "Global".BUTTON_Led_Test)
   END_RUNG
   // the same network as SCL:
   "Button_sound_off"(input := "DIa1.5",   // "DI_Single"
                      delay_time := "Preset_values".DI_timer_delay_time_slow,
                      filter := true,
                      value => "Global".BUTTON_Sound_Off,
                      ENO => #_w1);
   "Button_global_stop"(EN := #_w1,   // "DI_Single"
                        input := "DIa1.6",
                        delay_time := "Preset_values".DI_timer_delay_time_superfast,
                        filter := true,
                        value => "Global".BUTTON_Global_Stop,
                        ENO => #_w2);
   IF #_w2 THEN
       "Button_led_test"(input := "DIb1.1",   // "DI_Single"
                         delay_time := "Preset_values".DI_timer_delay_time_superfast,
                         filter := true,
                         value => "Global".BUTTON_Led_Test);
   END_IF;
END_REGION

